C03625=1054.668,133.483,-83.506,171.485,33.116,156.194
C03626=1054.674,133.732,-83.526,171.487,33.118,156.195
C03627=1054.680,133.981,-83.548,171.489,33.121,156.195
C03628=1054.685,134.230,-83.568,171.490,33.123,156.195
C03629=1054.692,134.479,-83.589,171.492,33.125,156.196
C03630=1054.698,134.728,-83.610,171.494,33.128,156.196
C03631=1054.704,134.977,-83.632,171.496,33.130,156.197
C03632=1054.710,135.226,-83.652,171.498,33.132,156.197
C03633=1054.716,135.475,-83.673,171.499,33.135,156.197
C03634=1054.721,135.724,-83.694,171.501,33.137,156.198
C03635=1054.728,135.973,-83.715,171.503,33.139,156.198
C03636=1054.733,136.222,-83.735,171.505,33.142,156.199
C03637=1054.739,136.471,-83.757,171.507,33.145,156.199
C03638=1054.746,136.720,-83.778,171.508,33.146,156.199
C03639=1054.752,136.969,-83.799,171.510,33.149,156.200
C03640=1054.758,137.219,-83.820,171.512,33.152,156.200
C03641=1054.764,137.468,-83.840,171.514,33.154,156.201
C03642=1054.770,137.717,-83.862,171.516,33.156,156.201
C03643=1054.776,137.965,-83.883,171.518,33.159,156.201
C03644=1054.781,138.215,-83.904,171.519,33.161,156.202
C03645=1054.788,138.463,-83.925,171.521,33.163,156.202
C03646=1054.794,138.712,-83.946,171.523,33.166,156.203
C03647=1054.800,138.962,-83.967,171.525,33.168,156.203
C03648=1054.805,139.211,-83.989,171.527,33.170,156.203
C03649=1054.812,139.460,-84.010,171.528,33.173,156.204
C03650=1054.817,139.709,-84.030,171.530,33.175,156.204
C03651=1054.824,139.958,-84.052,171.532,33.178,156.205
C03652=1054.830,140.207,-84.073,171.534,33.180,156.205
C03653=1054.835,140.456,-84.094,171.536,33.183,156.205
C03654=1054.841,140.706,-84.116,171.538,33.185,156.206
C03655=1054.847,140.954,-84.137,171.539,33.188,156.206
C03656=1054.854,141.203,-84.158,171.541,33.190,156.207
C03657=1054.859,141.451,-84.179,171.543,33.192,156.207
C03658=1054.865,141.701,-84.200,171.545,33.195,156.207
C03659=1054.871,141.964,-84.223,171.547,33.197,156.208
C03660=1054.878,142.228,-84.246,171.549,33.200,156.208
C03661=1054.884,142.491,-84.268,171.551,33.203,156.209
C03662=1054.890,142.754,-84.291,171.553,33.205,156.209
C03663=1054.895,143.004,-84.312,171.554,33.208,156.210
C03664=1054.902,143.253,-84.333,171.556,33.210,156.210
C03665=1054.908,143.502,-84.355,171.558,33.212,156.210
C03666=1054.913,143.750,-84.376,171.560,33.215,156.211
C03667=1054.920,143.999,-84.397,171.562,33.217,156.211
C03668=1054.926,144.249,-84.419,171.564,33.220,156.212
C03669=1054.932,144.497,-84.440,171.566,33.222,156.212
C03670=1054.938,144.747,-84.461,171.567,33.224,156.212
C03671=1054.944,144.996,-84.483,171.569,33.227,156.213
C03672=1054.950,145.245,-84.504,171.571,33.229,156.213
C03673=1054.956,145.494,-84.526,171.573,33.231,156.214
C03674=1054.962,145.743,-84.547,171.575,33.234,156.214
C03675=1054.967,145.991,-84.568,171.577,33.237,156.214
C03676=1054.974,146.241,-84.590,171.579,33.239,156.215
C03677=1054.980,146.490,-84.612,171.580,33.241,156.215
C03678=1054.985,146.738,-84.633,171.582,33.244,156.216
C03679=1054.992,146.988,-84.655,171.584,33.246,156.216
C03680=1054.998,147.237,-84.676,171.586,33.249,156.217
C03681=1055.003,147.485,-84.698,171.588,33.251,156.217
C03682=1055.009,147.735,-84.719,171.590,33.253,156.217
C03683=1055.016,147.984,-84.741,171.592,33.256,156.218
C03684=1055.022,148.233,-84.762,171.593,33.258,156.218
C03685=1055.027,148.481,-84.784,171.595,33.261,156.219
C03686=1055.033,148.731,-84.805,171.597,33.263,156.219
C03687=1055.040,148.980,-84.827,171.599,33.266,156.219
C03688=1055.045,149.228,-84.848,171.601,33.268,156.220
C03689=1055.051,149.478,-84.870,171.603,33.271,156.220
C03690=1055.057,149.727,-84.892,171.605,33.273,156.221
C03691=1055.063,149.976,-84.914,171.607,33.276,156.221
C03692=1055.069,150.224,-84.936,171.608,33.278,156.221
C03693=1055.075,150.473,-84.957,171.610,33.280,156.222
C03694=1055.081,150.723,-84.979,171.612,33.283,156.222
C03695=1055.087,150.971,-85.000,171.614,33.285,156.223
C03696=1055.093,151.220,-85.022,171.616,33.288,156.223
C03697=1055.098,151.470,-85.044,171.618,33.291,156.224
C03698=1055.104,151.719,-85.066,171.620,33.292,156.224
C03699=1055.110,151.967,-85.088,171.622,33.295,156.224
C03700=1055.116,152.216,-85.109,171.624,33.298,156.225
C03701=1055.123,152.465,-85.131,171.625,33.300,156.225
C03702=1055.128,152.715,-85.153,171.627,33.303,156.226
C03703=1055.134,152.963,-85.175,171.629,33.305,156.226
C03704=1055.140,153.212,-85.197,171.632,33.308,156.227
C03705=1055.146,153.461,-85.219,171.634,33.310,156.227
C03706=1055.152,153.710,-85.240,171.636,33.312,156.227
C03707=1055.158,153.960,-85.262,171.638,33.315,156.228
C03708=1055.164,154.208,-85.284,171.640,33.317,156.228
C03709=1055.170,154.457,-85.306,171.642,33.320,156.229
C03710=1055.176,154.706,-85.328,171.644,33.323,156.229
C03711=1055.181,154.956,-85.350,171.645,33.324,156.229
C03712=1055.188,155.204,-85.372,171.647,33.327,156.230
C03713=1055.193,155.453,-85.394,171.649,33.330,156.230
C03714=1055.200,155.702,-85.415,171.651,33.332,156.231
C03715=1055.205,155.951,-85.438,171.653,33.335,156.231
C03716=1055.212,156.200,-85.460,171.655,33.337,156.232
C03717=1055.218,156.449,-85.481,171.657,33.340,156.232
C03718=1055.223,156.698,-85.504,171.659,33.342,156.233
C03719=1055.229,156.947,-85.526,171.661,33.345,156.233
C03720=1055.235,157.196,-85.549,171.663,33.348,156.233
C03721=1055.241,157.445,-85.570,171.665,33.350,156.234
C03722=1055.247,157.694,-85.592,171.667,33.352,156.234
C03723=1055.254,157.978,-85.617,171.669,33.355,156.235
C03724=1055.261,158.263,-85.642,171.671,33.358,156.235
C03725=1055.267,158.548,-85.668,171.673,33.361,156.236
C03726=1055.274,158.833,-85.693,171.675,33.364,156.236
C03727=1055.280,159.082,-85.715,171.677,33.366,156.237
C03728=1055.286,159.331,-85.738,171.679,33.369,156.237
C03729=1055.292,159.580,-85.760,171.681,33.371,156.237
C03730=1055.299,159.829,-85.782,171.683,33.374,156.238
C03731=1055.304,160.077,-85.804,171.685,33.376,156.238
C03732=1055.310,160.326,-85.826,171.687,33.379,156.239
C03733=1055.316,160.575,-85.849,171.689,33.381,156.239
C03734=1055.322,160.824,-85.870,171.691,33.383,156.240
C03735=1055.327,161.073,-85.893,171.693,33.387,156.240
C03736=1055.334,161.323,-85.915,171.695,33.389,156.241
C03737=1055.339,161.571,-85.938,171.697,33.392,156.241
C03738=1055.345,161.820,-85.961,171.699,33.394,156.241
C03739=1055.350,162.069,-85.983,171.701,33.397,156.242
C03740=1055.356,162.318,-86.005,171.703,33.399,156.242
C03741=1055.362,162.567,-86.028,171.705,33.402,156.243
C03742=1055.367,162.816,-86.050,171.706,33.404,156.243
C03743=1055.374,163.065,-86.073,171.708,33.407,156.244
C03744=1055.380,163.314,-86.096,171.710,33.410,156.244
C03745=1055.385,163.563,-86.118,171.712,33.413,156.245
C03746=1055.390,163.811,-86.140,171.714,33.415,156.245
C03747=1055.397,164.060,-86.163,171.716,33.418,156.245
C03748=1055.402,164.309,-86.185,171.718,33.420,156.246
C03749=1055.408,164.558,-86.208,171.720,33.423,156.246
C03750=1055.414,164.807,-86.231,171.723,33.425,156.247
C03751=1055.420,165.056,-86.253,171.725,33.428,156.247
C03752=1055.426,165.305,-86.275,171.727,33.431,156.248
C03753=1055.431,165.554,-86.298,171.729,33.433,156.248
C03754=1055.437,165.803,-86.321,171.731,33.436,156.249
C03755=1055.443,166.051,-86.343,171.733,33.439,156.249
C03756=1055.448,166.301,-86.366,171.735,33.441,156.250
C03757=1055.454,166.549,-86.389,171.737,33.444,156.250
C03758=1055.460,166.798,-86.411,171.739,33.446,156.250
C03759=1055.465,167.047,-86.434,171.741,33.449,156.251
C03760=1055.472,167.296,-86.457,171.743,33.452,156.251
C03761=1055.477,167.545,-86.479,171.745,33.454,156.252
C03762=1055.483,167.794,-86.502,171.747,33.457,156.252
C03763=1055.489,168.043,-86.525,171.749,33.459,156.253
C03764=1055.495,168.292,-86.547,171.751,33.462,156.253
C03765=1055.501,168.541,-86.570,171.753,33.465,156.254
C03766=1055.507,168.789,-86.593,171.755,33.468,156.254
C03767=1055.512,169.038,-86.616,171.757,33.470,156.255
C03768=1055.518,169.288,-86.638,171.759,33.473,156.255
C03769=1055.524,169.536,-86.661,171.761,33.475,156.255
C03770=1055.530,169.785,-86.684,171.763,33.478,156.256
C03771=1055.536,170.034,-86.707,171.765,33.480,156.256
C03772=1055.542,170.283,-86.729,171.767,33.483,156.257
C03773=1055.547,170.532,-86.752,171.769,33.485,156.257
C03774=1055.554,170.781,-86.775,171.771,33.488,156.258
C03775=1055.559,171.030,-86.798,171.773,33.491,156.258
C03776=1055.565,171.278,-86.821,171.775,33.494,156.259
C03777=1055.571,171.527,-86.844,171.777,33.496,156.259
C03778=1055.577,171.776,-86.867,171.779,33.499,156.260
C03779=1055.583,172.025,-86.889,171.781,33.501,156.260
C03780=1055.589,172.274,-86.912,171.783,33.504,156.260
C03781=1055.595,172.523,-86.935,171.785,33.506,156.261
C03782=1055.601,172.772,-86.958,171.788,33.509,156.261
C03783=1055.607,173.021,-86.981,171.790,33.511,156.262
C03784=1055.612,173.270,-87.004,171.792,33.514,156.262
C03785=1055.619,173.519,-87.026,171.794,33.517,156.263
C03786=1055.625,173.767,-87.049,171.796,33.520,156.263
C03787=1055.631,174.052,-87.076,171.798,33.522,156.264
C03788=1055.638,174.336,-87.102,171.801,33.525,156.264
C03789=1055.645,174.620,-87.128,171.803,33.529,156.265
C03790=1055.651,174.905,-87.155,171.805,33.531,156.265
C03791=1055.657,175.154,-87.178,171.808,33.534,156.266
C03792=1055.664,175.403,-87.200,171.810,33.537,156.266
C03793=1055.670,175.651,-87.224,171.812,33.539,156.267
C03794=1055.676,175.900,-87.247,171.814,33.542,156.267
C03795=1055.682,176.149,-87.270,171.816,33.545,156.267
C03796=1055.687,176.398,-87.293,171.818,33.547,156.268
C03797=1055.693,176.647,-87.316,171.820,33.550,156.268
C03798=1055.699,176.896,-87.339,171.822,33.552,156.269
C03799=1055.705,177.145,-87.363,171.824,33.555,156.269
C03800=1055.712,177.393,-87.385,171.826,33.558,156.270
C03801=1055.718,177.642,-87.408,171.828,33.560,156.270
C03802=1055.723,177.891,-87.431,171.830,33.563,156.271
C03803=1055.730,178.140,-87.455,171.832,33.565,156.271
C03804=1055.736,178.389,-87.478,171.834,33.568,156.272
C03805=1055.741,178.638,-87.501,171.837,33.571,156.272
C03806=1055.747,178.887,-87.524,171.839,33.573,156.272
C03807=1055.753,179.135,-87.548,171.841,33.576,156.273
C03808=1055.760,179.384,-87.570,171.844,33.579,156.273
C03809=1055.766,179.633,-87.593,171.846,33.581,156.274
C03810=1055.772,179.881,-87.617,171.848,33.584,156.274
C03811=1055.778,180.130,-87.640,171.850,33.586,156.275
C03812=1055.784,180.380,-87.663,171.852,33.589,156.275
C03813=1055.790,180.628,-87.687,171.854,33.592,156.276
C03814=1055.796,180.877,-87.710,171.856,33.594,156.276
C03815=1055.802,181.126,-87.733,171.859,33.597,156.277
C03816=1055.808,181.375,-87.757,171.861,33.600,156.277
C03817=1055.814,181.624,-87.780,171.863,33.602,156.278
C03818=1055.820,181.873,-87.803,171.865,33.605,156.278
C03819=1055.827,182.121,-87.826,171.867,33.607,156.278
C03820=1055.833,182.370,-87.849,171.869,33.610,156.279
C03821=1055.839,182.619,-87.873,171.871,33.613,156.279
C03822=1055.845,182.868,-87.896,171.873,33.615,156.280
C03823=1055.851,183.116,-87.920,171.876,33.618,156.280
C03824=1055.857,183.365,-87.943,171.878,33.621,156.281
C03825=1055.863,183.615,-87.966,171.880,33.623,156.281
C03826=1055.869,183.863,-87.989,171.882,33.626,156.282
C03827=1055.875,184.112,-88.012,171.884,33.628,156.282
C03828=1055.882,184.361,-88.036,171.886,33.631,156.283
C03829=1055.887,184.610,-88.059,171.888,33.634,156.283
C03830=1055.893,184.859,-88.084,171.892,33.637,156.284
C03831=1055.899,185.107,-88.107,171.894,33.640,156.284
C03832=1055.904,185.357,-88.131,171.896,33.642,156.285
C03833=1055.910,185.605,-88.155,171.898,33.645,156.285
C03834=1055.916,185.854,-88.179,171.900,33.648,156.286
C03835=1055.921,186.102,-88.202,171.902,33.651,156.286
C03836=1055.928,186.351,-88.226,171.904,33.654,156.287
C03837=1055.933,186.600,-88.250,171.906,33.656,156.287
C03838=1055.939,186.849,-88.273,171.909,33.659,156.288
C03839=1055.944,187.098,-88.298,171.911,33.662,156.288
C03840=1055.951,187.347,-88.322,171.913,33.664,156.288
C03841=1055.956,187.596,-88.345,171.915,33.668,156.289
C03842=1055.962,187.844,-88.369,171.917,33.670,156.289
C03843=1055.969,188.093,-88.393,171.919,33.673,156.290
C03844=1055.974,188.342,-88.416,171.921,33.676,156.290
C03845=1055.980,188.590,-88.440,171.923,33.679,156.291
C03846=1055.986,188.840,-88.465,171.926,33.682,156.291
C03847=1055.992,189.088,-88.488,171.928,33.685,156.292
C03848=1055.997,189.337,-88.513,171.931,33.687,156.292
C03849=1056.003,189.586,-88.536,171.933,33.690,156.293
C03850=1056.009,189.835,-88.560,171.935,33.693,156.294
C03851=1056.015,190.118,-88.588,171.938,33.696,156.294
C03852=1056.022,190.402,-88.615,171.940,33.699,156.295
C03853=1056.028,190.687,-88.642,171.943,33.702,156.295
C03854=1056.035,190.970,-88.670,171.945,33.705,156.296
C03855=1056.042,191.219,-88.694,171.947,33.709,156.296
C03856=1056.047,191.468,-88.718,171.950,33.711,156.297
C03857=1056.054,191.717,-88.742,171.952,33.714,156.297
C03858=1056.059,191.966,-88.765,171.954,33.717,156.298
C03859=1056.065,192.214,-88.789,171.956,33.720,156.298
C03860=1056.071,192.463,-88.813,171.958,33.722,156.299
C03861=1056.077,192.712,-88.837,171.960,33.726,156.299
C03862=1056.083,192.961,-88.861,171.963,33.728,156.300
C03863=1056.088,193.209,-88.886,171.965,33.731,156.300
C03864=1056.095,193.458,-88.909,171.967,33.734,156.301
C03865=1056.100,193.707,-88.934,171.970,33.737,156.301
C03866=1056.106,193.955,-88.958,171.972,33.739,156.302
C03867=1056.112,194.204,-88.982,171.975,33.742,156.302
C03868=1056.118,194.453,-89.006,171.977,33.745,156.303
C03869=1056.124,194.702,-89.030,171.979,33.748,156.303
C03870=1056.130,194.951,-89.055,171.981,33.751,156.304
C03871=1056.136,195.200,-89.079,171.984,33.753,156.304
C03872=1056.142,195.448,-89.103,171.986,33.757,156.305
C03873=1056.148,195.697,-89.127,171.988,33.759,156.305
C03874=1056.153,195.946,-89.151,171.990,33.762,156.306
C03875=1056.160,196.195,-89.175,171.992,33.765,156.306
C03876=1056.165,196.443,-89.200,171.995,33.768,156.307
C03877=1056.172,196.692,-89.224,171.997,33.771,156.307
C03878=1056.177,196.941,-89.248,171.999,33.774,156.308
C03879=1056.184,197.189,-89.273,172.001,33.777,156.308
C03880=1056.190,197.438,-89.297,172.005,33.779,156.309
C03881=1056.196,197.687,-89.321,172.007,33.782,156.309
C03882=1056.202,197.935,-89.345,172.009,33.785,156.310
C03883=1056.208,198.184,-89.369,172.011,33.788,156.310
C03884=1056.214,198.434,-89.394,172.014,33.791,156.311
C03885=1056.220,198.682,-89.419,172.016,33.794,156.311
C03886=1056.226,198.931,-89.443,172.018,33.796,156.312
C03887=1056.232,199.179,-89.467,172.020,33.799,156.312
C03888=1056.238,199.428,-89.491,172.023,33.802,156.313
C03889=1056.244,199.677,-89.515,172.025,33.805,156.313
C03890=1056.250,199.925,-89.540,172.027,33.808,156.314
C03891=1056.256,200.174,-89.565,172.030,33.811,156.314
C03892=1056.262,200.423,-89.589,172.032,33.813,156.315
C03893=1056.268,200.672,-89.613,172.034,33.816,156.316
C03894=1056.275,200.921,-89.638,172.037,33.819,156.316
C03895=1056.281,201.169,-89.662,172.040,33.822,156.317
C03896=1056.286,201.418,-89.687,172.042,33.825,156.317
C03897=1056.292,201.666,-89.712,172.044,33.828,156.318
C03898=1056.299,201.915,-89.736,172.047,33.831,156.318
C03899=1056.305,202.164,-89.760,172.049,33.834,156.319
C03900=1056.310,202.412,-89.785,172.051,33.836,156.319
C03901=1056.316,202.662,-89.810,172.053,33.840,156.320
C03902=1056.321,202.910,-89.834,172.056,33.843,156.320
C03903=1056.328,203.159,-89.859,172.058,33.845,156.321
C03904=1056.334,203.408,-89.883,172.060,33.848,156.321
C03905=1056.340,203.656,-89.908,172.063,33.852,156.322
C03906=1056.346,203.905,-89.933,172.065,33.855,156.322
C03907=1056.352,204.154,-89.958,172.067,33.857,156.323
C03908=1056.357,204.402,-89.983,172.070,33.860,156.323
C03909=1056.363,204.651,-90.008,172.073,33.863,156.324
C03910=1056.369,204.900,-90.032,172.075,33.866,156.325
C03911=1056.375,205.148,-90.058,172.077,33.870,156.325
C03912=1056.382,205.397,-90.082,172.080,33.872,156.326
C03913=1056.387,205.645,-90.107,172.082,33.875,156.326
C03914=1056.393,205.895,-90.131,172.084,33.878,156.327
C03915=1056.418,206.946,-90.237,172.283,33.968,156.339
C03916=1056.424,207.183,-90.261,172.285,33.972,156.340
C03917=1056.431,207.420,-90.286,172.287,33.975,156.341
C03918=1056.437,207.658,-90.310,172.288,33.979,156.342
C03919=1056.442,207.895,-90.336,172.291,33.983,156.342
C03920=1056.448,208.133,-90.360,172.293,33.986,156.343
C03921=1056.454,208.371,-90.384,172.295,33.990,156.344
C03922=1056.460,208.607,-90.409,172.296,33.993,156.344
C03923=1056.466,208.846,-90.434,172.298,33.997,156.345
C03924=1056.472,209.094,-90.460,172.300,34.001,156.346
C03925=1056.479,209.342,-90.485,172.302,34.005,156.347
C03926=1056.484,209.591,-90.512,172.304,34.009,156.347
C03927=1056.491,209.840,-90.537,172.306,34.013,156.348
C03928=1056.498,210.088,-90.564,172.308,34.017,156.349
C03929=1056.504,210.337,-90.589,172.310,34.020,156.349
C03930=1056.510,210.585,-90.616,172.312,34.024,156.350
C03931=1056.516,210.834,-90.641,172.314,34.028,156.351
C03932=1056.522,211.082,-90.667,172.315,34.032,156.352
C03933=1056.528,211.332,-90.693,172.317,34.035,156.352
C03934=1056.535,211.580,-90.719,172.320,34.040,156.353
C03935=1056.541,211.828,-90.745,172.322,34.043,156.354
C03936=1056.547,212.077,-90.771,172.324,34.047,156.355
C03937=1056.554,212.325,-90.798,172.326,34.051,156.355
C03938=1056.559,212.574,-90.824,172.327,34.055,156.356
C03939=1056.566,212.822,-90.850,172.329,34.058,156.357
C03940=1056.571,213.071,-90.876,172.332,34.062,156.358
C03941=1056.578,213.320,-90.902,172.334,34.066,156.358
C03942=1056.584,213.569,-90.929,172.336,34.070,156.359
C03943=1056.591,213.817,-90.954,172.338,34.074,156.360
C03944=1056.596,214.066,-90.981,172.339,34.078,156.361
C03945=1056.603,214.314,-91.007,172.341,34.081,156.361
C03946=1056.609,214.562,-91.033,172.343,34.085,156.362
C03947=1056.615,214.811,-91.059,172.346,34.089,156.363
C03948=1056.621,215.060,-91.086,172.348,34.093,156.363
C03949=1056.628,215.308,-91.112,172.350,34.097,156.364
C03950=1056.633,215.556,-91.138,172.352,34.100,156.365
C03951=1056.640,215.806,-91.164,172.354,34.104,156.366
C03952=1056.646,216.054,-91.191,172.355,34.108,156.366
C03953=1056.653,216.302,-91.217,172.357,34.112,156.367
C03954=1056.659,216.551,-91.244,172.360,34.115,156.368
C03955=1056.665,216.800,-91.269,172.362,34.119,156.368
C03956=1056.671,217.048,-91.296,172.364,34.123,156.369
C03957=1056.677,217.296,-91.322,172.366,34.127,156.370
C03958=1056.684,217.545,-91.349,172.368,34.130,156.371
C03959=1056.690,217.794,-91.376,172.370,34.134,156.371
C03960=1056.696,218.042,-91.402,172.373,34.138,156.372
C03961=1056.702,218.291,-91.428,172.374,34.142,156.373
C03962=1056.709,218.539,-91.454,172.376,34.146,156.374
C03963=1056.714,218.788,-91.481,172.378,34.149,156.374
C03964=1056.722,219.036,-91.507,172.380,34.153,156.375
C03965=1056.727,219.285,-91.534,172.382,34.156,156.376
C03966=1056.734,219.533,-91.560,172.384,34.161,156.377
C03967=1056.740,219.782,-91.587,172.387,34.164,156.377
C03968=1056.746,220.030,-91.613,172.389,34.168,156.378
C03969=1056.753,220.279,-91.640,172.391,34.172,156.379
C03970=1056.759,220.527,-91.666,172.393,34.175,156.379
C03971=1056.765,220.775,-91.692,172.395,34.179,156.380
C03972=1056.771,221.016,-91.718,172.397,34.183,156.381
C03973=1056.777,221.256,-91.744,172.399,34.186,156.382
C03974=1056.783,221.496,-91.769,172.401,34.190,156.382
C03975=1056.789,221.736,-91.795,172.403,34.194,156.383
C03976=1056.795,221.976,-91.822,172.405,34.198,156.384
C03977=1056.801,222.217,-91.847,172.407,34.201,156.384
C03978=1056.808,222.457,-91.873,172.409,34.205,156.385
C03979=1056.813,222.697,-91.899,172.412,34.209,156.386
C03980=1056.819,222.945,-91.926,172.413,34.212,156.387
C03981=1056.825,223.193,-91.952,172.415,34.216,156.387
C03982=1056.831,223.442,-91.979,172.417,34.219,156.388
C03983=1056.837,223.691,-92.006,172.419,34.223,156.389
C03984=1056.844,223.940,-92.032,172.421,34.227,156.389
C03985=1056.850,224.188,-92.059,172.424,34.231,156.390
C03986=1056.857,224.436,-92.087,172.426,34.235,156.391
C03987=1056.863,224.685,-92.113,172.428,34.238,156.392
C03988=1056.868,224.933,-92.140,172.430,34.242,156.392
C03989=1056.875,225.182,-92.167,172.432,34.246,156.393
C03990=1056.881,225.430,-92.193,172.434,34.250,156.394
C03991=1056.888,225.679,-92.221,172.437,34.253,156.395
C03992=1056.894,225.927,-92.248,172.439,34.257,156.395
C03993=1056.900,226.176,-92.275,172.441,34.261,156.396
C03994=1056.906,226.424,-92.301,172.443,34.264,156.397
C03995=1056.912,226.673,-92.329,172.445,34.268,156.397
C03996=1056.919,226.921,-92.355,172.447,34.272,156.398
C03997=1056.925,227.170,-92.382,172.450,34.276,156.399
C03998=1056.931,227.418,-92.409,172.452,34.279,156.400
C03999=1056.938,227.667,-92.436,172.454,34.283,156.400
C04000=1056.944,227.915,-92.463,172.456,34.287,156.401
C04001=1056.950,228.164,-92.491,172.458,34.290,156.402
C04002=1056.956,228.412,-92.517,172.460,34.294,156.402
C04003=1056.963,228.661,-92.544,172.463,34.298,156.403
C04004=1056.969,228.908,-92.571,172.465,34.302,156.404
C04005=1056.976,229.157,-92.598,172.467,34.305,156.405
C04006=1056.981,229.406,-92.625,172.469,34.309,156.405
C04007=1056.988,229.654,-92.653,172.471,34.313,156.406
C04008=1056.994,229.903,-92.679,172.473,34.316,156.407
C04009=1057.001,230.151,-92.707,172.476,34.320,156.407
C04010=1057.006,230.399,-92.734,172.478,34.324,156.408
C04011=1057.013,230.648,-92.761,172.480,34.328,156.409
C04012=1057.019,230.897,-92.789,172.482,34.331,156.410
C04013=1057.025,231.145,-92.816,172.484,34.335,156.410
C04014=1057.031,231.394,-92.843,172.487,34.339,156.411
C04015=1057.037,231.642,-92.871,172.489,34.342,156.412
C04016=1057.044,231.891,-92.898,172.491,34.346,156.413
C04017=1057.050,232.139,-92.925,172.493,34.350,156.413
C04018=1057.056,232.388,-92.952,172.495,34.354,156.414
C04019=1057.062,232.635,-92.979,172.497,34.357,156.415
C04020=1057.068,232.884,-93.006,172.500,34.361,156.416
C04021=1057.075,233.133,-93.034,172.502,34.364,156.416
C04022=1057.080,233.381,-93.062,172.504,34.368,156.417
C04023=1057.087,233.630,-93.089,172.506,34.372,156.418
C04024=1057.093,233.878,-93.117,172.508,34.376,156.418
C04025=1057.100,234.126,-93.144,172.512,34.380,156.419
C04026=1057.105,234.375,-93.172,172.514,34.383,156.420
C04027=1057.111,234.623,-93.199,172.516,34.387,156.421
C04028=1057.117,234.860,-93.225,172.518,34.390,156.421
C04029=1057.124,235.096,-93.252,172.520,34.394,156.422
C04030=1057.129,235.332,-93.278,172.522,34.398,156.423
C04031=1057.135,235.568,-93.304,172.524,34.401,156.423
C04032=1057.141,235.804,-93.330,172.526,34.405,156.424
C04033=1057.147,236.041,-93.357,172.528,34.408,156.425
C04034=1057.153,236.277,-93.382,172.530,34.412,156.425
C04035=1057.159,236.513,-93.409,172.532,34.415,156.426
C04036=1057.165,236.762,-93.436,172.535,34.419,156.427
C04037=1057.171,237.010,-93.464,172.538,34.422,156.428
C04038=1057.177,237.258,-93.491,172.540,34.426,156.428
C04039=1057.184,237.507,-93.519,172.542,34.430,156.429
C04040=1057.190,237.754,-93.547,172.544,34.434,156.430
C04041=1057.196,238.003,-93.575,172.546,34.437,156.430
C04042=1057.202,238.252,-93.602,172.549,34.441,156.431
C04043=1057.208,238.500,-93.629,172.551,34.445,156.432
C04044=1057.215,238.748,-93.657,172.553,34.448,156.433
C04045=1057.221,238.997,-93.685,172.555,34.452,156.433
C04046=1057.228,239.245,-93.713,172.557,34.456,156.434
C04047=1057.234,239.493,-93.740,172.561,34.459,156.435
C04048=1057.240,239.742,-93.769,172.563,34.463,156.435
C04049=1057.246,239.990,-93.796,172.565,34.466,156.436
C04050=1057.253,240.239,-93.824,172.567,34.471,156.437
C04051=1057.258,240.487,-93.852,172.569,34.474,156.438
C04052=1057.265,240.735,-93.880,172.572,34.478,156.438
C04053=1057.272,240.984,-93.908,172.574,34.481,156.439
C04054=1057.278,241.233,-93.936,172.576,34.485,156.440
C04055=1057.284,241.480,-93.963,172.579,34.489,156.441
C04056=1057.290,241.729,-93.991,172.581,34.492,156.441
C04057=1057.296,241.977,-94.019,172.584,34.496,156.442
C04058=1057.303,242.226,-94.047,172.586,34.500,156.443
C04059=1057.308,242.474,-94.075,172.588,34.503,156.443
C04060=1057.315,242.722,-94.103,172.590,34.507,156.444
C04061=1057.321,242.971,-94.131,172.592,34.511,156.445
C04062=1057.327,243.220,-94.159,172.596,34.515,156.446
C04063=1057.333,243.468,-94.187,172.598,34.518,156.446
C04064=1057.339,243.716,-94.215,172.600,34.522,156.447
C04065=1057.346,243.964,-94.244,172.602,34.525,156.448
C04066=1057.352,244.213,-94.272,172.604,34.529,156.448
C04067=1057.358,244.461,-94.299,172.607,34.533,156.449
C04068=1057.364,244.709,-94.328,172.609,34.537,156.450
C04069=1057.370,244.958,-94.356,172.612,34.540,156.451
C04070=1057.377,245.206,-94.384,172.614,34.544,156.451
C04071=1057.383,245.455,-94.413,172.616,34.548,156.452
C04072=1057.390,245.703,-94.440,172.619,34.551,156.453
C04073=1057.395,245.951,-94.468,172.621,34.555,156.454
C04074=1057.401,246.200,-94.497,172.623,34.558,156.454
C04075=1057.408,246.448,-94.525,172.626,34.563,156.455
C04076=1057.414,246.697,-94.553,172.628,34.566,156.456
C04077=1057.420,246.945,-94.582,172.631,34.570,156.457
C04078=1057.425,247.193,-94.610,172.633,34.574,156.457
C04079=1057.432,247.441,-94.638,172.635,34.577,156.458
C04080=1057.438,247.689,-94.667,172.637,34.581,156.459
C04081=1057.444,247.938,-94.696,172.641,34.585,156.460
C04082=1057.450,248.187,-94.724,172.643,34.589,156.460
C04083=1057.456,248.434,-94.753,172.645,34.592,156.461
C04084=1057.462,248.668,-94.779,172.647,34.596,156.462
C04085=1057.468,248.901,-94.806,172.649,34.599,156.462
C04086=1057.473,249.134,-94.833,172.652,34.603,156.463
C04087=1057.479,249.367,-94.859,172.654,34.607,156.464
C04088=1057.485,249.600,-94.886,172.656,34.610,156.464
C04089=1057.491,249.834,-94.912,172.658,34.613,156.465
C04090=1057.496,250.067,-94.940,172.660,34.617,156.466
C04091=1057.502,250.300,-94.967,172.664,34.620,156.467
C04092=1057.508,250.548,-94.995,172.666,34.624,156.467
C04093=1057.514,250.797,-95.024,172.668,34.628,156.468
C04094=1057.520,251.045,-95.052,172.670,34.631,156.469
C04095=1057.527,251.293,-95.081,172.672,34.635,156.469
C04096=1057.533,251.542,-95.109,172.676,34.639,156.470
C04097=1057.539,251.789,-95.138,172.678,34.643,156.471
C04098=1057.545,252.037,-95.167,172.680,34.646,156.472
C04099=1057.551,252.286,-95.195,172.682,34.650,156.472
C04100=1057.557,252.534,-95.224,172.686,34.653,156.473
C04101=1057.563,252.783,-95.253,172.688,34.657,156.474
C04102=1057.570,253.031,-95.281,172.690,34.661,156.475
C04103=1057.577,253.279,-95.310,172.692,34.665,156.475
C04104=1057.583,253.528,-95.338,172.695,34.668,156.476
C04105=1057.589,253.776,-95.367,172.698,34.672,156.477
C04106=1057.595,254.024,-95.396,172.700,34.676,156.478
C04107=1057.601,254.273,-95.425,172.702,34.679,156.478
C04108=1057.607,254.521,-95.454,172.705,34.683,156.479
C04109=1057.613,254.769,-95.483,172.708,34.686,156.480
C04110=1057.620,255.017,-95.512,172.710,34.690,156.480
C04111=1057.626,255.266,-95.540,172.712,34.694,156.481
C04112=1057.633,255.514,-95.569,172.715,34.698,156.482
C04113=1057.639,255.762,-95.598,172.717,34.701,156.483
C04114=1057.645,256.010,-95.627,172.720,34.705,156.483
C04115=1057.651,256.258,-95.656,172.723,34.709,156.484
C04116=1057.657,256.507,-95.684,172.725,34.712,156.485
C04117=1057.664,256.755,-95.713,172.727,34.716,156.486
C04118=1057.670,257.003,-95.742,172.730,34.719,156.486
C04119=1057.676,257.251,-95.771,172.733,34.723,156.487
C04120=1057.683,257.500,-95.801,172.735,34.727,156.488
C04121=1057.689,257.748,-95.830,172.737,34.730,156.488
C04122=1057.696,257.997,-95.857,172.740,34.734,156.489
C04123=1057.702,258.245,-95.886,172.743,34.738,156.490
C04124=1057.708,258.493,-95.915,172.745,34.741,156.491
C04125=1057.715,258.741,-95.944,172.748,34.745,156.491
C04126=1057.721,258.989,-95.974,172.750,34.749,156.492
C04127=1057.727,259.237,-96.003,172.753,34.752,156.493
C04128=1057.733,259.485,-96.032,172.756,34.756,156.494
C04129=1057.740,259.734,-96.061,172.758,34.759,156.494
C04130=1057.746,259.982,-96.090,172.760,34.763,156.495
C04131=1057.753,260.231,-96.119,172.764,34.767,156.496
C04132=1057.759,260.479,-96.148,172.766,34.770,156.496
C04133=1057.765,260.727,-96.177,172.768,34.774,156.497
C04134=1057.771,260.975,-96.206,172.771,34.777,156.498
C04135=1057.778,261.224,-96.236,172.773,34.781,156.499
C04136=1057.785,261.472,-96.265,172.776,34.785,156.499
C04137=1057.791,261.720,-96.294,172.779,34.788,156.500
C04138=1057.797,261.968,-96.323,172.781,34.792,156.501
C04139=1057.803,262.216,-96.352,172.784,34.795,156.501
C04140=1057.810,262.448,-96.379,172.787,34.799,156.502
C04141=1057.816,262.680,-96.407,172.789,34.803,156.503
C04142=1057.822,262.912,-96.434,172.791,34.806,156.503
C04143=1057.828,263.145,-96.461,172.793,34.809,156.504
C04144=1057.834,263.378,-96.489,172.797,34.813,156.505
C04145=1057.840,263.610,-96.517,172.799,34.816,156.506
C04146=1057.846,263.841,-96.544,172.801,34.819,156.506
C04147=1057.851,264.073,-96.572,172.803,34.823,156.507
C04148=1057.857,264.321,-96.601,172.806,34.827,156.508
C04149=1057.864,264.570,-96.630,172.809,34.831,156.509
C04150=1057.870,264.819,-96.660,172.811,34.834,156.509
C04151=1057.876,265.066,-96.690,172.814,34.838,156.510
C04152=1057.882,265.314,-96.719,172.816,34.841,156.511
C04153=1057.888,265.563,-96.748,172.820,34.845,156.511
C04154=1057.895,265.811,-96.779,172.822,34.849,156.512
C04155=1057.901,266.059,-96.808,172.824,34.853,156.513
C04156=1057.907,266.308,-96.837,172.827,34.856,156.514
C04157=1057.913,266.555,-96.867,172.830,34.860,156.514
C04158=1057.920,266.804,-96.896,172.833,34.864,156.515
C04159=1057.926,267.052,-96.927,172.835,34.867,156.516
C04160=1057.932,267.300,-96.956,172.837,34.871,156.517
C04161=1057.939,267.548,-96.985,172.841,34.875,156.517
C04162=1057.945,267.797,-97.016,172.843,34.878,156.518
C04163=1057.951,268.045,-97.045,172.846,34.882,156.519
C04164=1057.958,268.292,-97.074,172.848,34.886,156.520
C04165=1057.963,268.541,-97.104,172.851,34.890,156.520
C04166=1057.971,268.789,-97.134,172.854,34.893,156.521
C04167=1057.976,269.037,-97.164,172.856,34.897,156.522
C04168=1057.983,269.285,-97.194,172.859,34.900,156.523
C04169=1057.989,269.534,-97.223,172.862,34.904,156.523
C04170=1057.995,269.781,-97.253,172.865,34.908,156.524
C04171=1058.002,270.029,-97.283,172.867,34.912,156.525
C04172=1058.008,270.278,-97.313,172.869,34.915,156.526
C04173=1058.014,270.526,-97.343,172.873,34.919,156.526
C04174=1058.020,270.774,-97.372,172.875,34.923,156.527
C04175=1058.027,271.022,-97.403,172.878,34.927,156.528
C04176=1058.033,271.270,-97.433,172.881,34.930,156.529
C04177=1058.039,271.518,-97.462,172.884,34.934,156.529
C04178=1058.046,271.767,-97.493,172.886,34.937,156.530
C04179=1058.052,272.014,-97.522,172.889,34.942,156.531
C04180=1058.058,272.262,-97.553,172.892,34.945,156.532
C04181=1058.065,272.511,-97.582,172.895,34.949,156.532
C04182=1058.071,272.759,-97.613,172.897,34.952,156.533
C04183=1058.076,273.007,-97.643,172.899,34.956,156.534
C04184=1058.084,273.255,-97.673,172.903,34.960,156.535
C04185=1058.089,273.503,-97.703,172.905,34.964,156.535
C04186=1058.095,273.751,-97.733,172.908,34.967,156.536
C04187=1058.102,273.999,-97.763,172.910,34.971,156.537
C04188=1058.108,274.247,-97.793,172.914,34.975,156.538
C04189=1058.115,274.495,-97.824,172.916,34.978,156.538
C04190=1058.121,274.743,-97.854,172.919,34.983,156.539
C04191=1058.126,274.991,-97.884,172.922,34.986,156.540
C04192=1058.134,275.240,-97.914,172.925,34.990,156.541
C04193=1058.139,275.488,-97.944,172.927,34.993,156.541
C04194=1058.146,275.736,-97.975,172.930,34.997,156.542
C04195=1058.152,275.984,-98.005,172.933,35.001,156.543
C04196=1058.158,276.218,-98.033,172.936,35.005,156.544
C04197=1058.163,276.452,-98.062,172.938,35.008,156.544
C04198=1058.170,276.686,-98.090,172.940,35.012,156.545
C04199=1058.176,276.920,-98.120,172.944,35.015,156.546
C04200=1058.182,277.155,-98.148,172.946,35.019,156.547
C04201=1058.188,277.388,-98.177,172.949,35.022,156.547
C04202=1058.193,277.623,-98.206,172.951,35.026,156.548
C04203=1058.200,277.857,-98.234,172.954,35.030,156.549
C04204=1058.206,278.105,-98.264,172.957,35.033,156.550
C04205=1058.212,278.353,-98.296,172.959,35.037,156.550
C04206=1058.218,278.601,-98.326,172.962,35.040,156.551
C04207=1058.225,278.849,-98.356,172.965,35.044,156.552
C04208=1058.231,279.097,-98.386,172.968,35.048,156.553
C04209=1058.237,279.345,-98.417,172.970,35.052,156.553
C04210=1058.243,279.593,-98.448,172.974,35.056,156.554
C04211=1058.250,279.841,-98.478,172.977,35.059,156.555
C04212=1058.256,280.089,-98.508,172.979,35.063,156.556
C04213=1058.263,280.337,-98.539,172.982,35.067,156.556
C04214=1058.269,280.585,-98.570,172.985,35.070,156.557
C04215=1058.275,280.833,-98.601,172.988,35.074,156.558
C04216=1058.281,281.081,-98.631,172.990,35.078,156.559
C04217=1058.288,281.329,-98.662,172.994,35.082,156.559
C04218=1058.294,281.577,-98.693,172.996,35.086,156.560
C04219=1058.300,281.825,-98.723,172.999,35.089,156.561
C04220=1058.306,282.073,-98.754,173.003,35.094,156.562
C04221=1058.313,282.321,-98.785,173.005,35.097,156.563
C04222=1058.318,282.569,-98.815,173.008,35.101,156.563
C04223=1058.325,282.817,-98.847,173.010,35.105,156.564
C04224=1058.332,283.065,-98.878,173.014,35.108,156.565
C04225=1058.337,283.313,-98.908,173.016,35.113,156.566
C04226=1058.344,283.561,-98.939,173.019,35.116,156.567
C04227=1058.350,283.809,-98.970,173.023,35.120,156.567
C04228=1058.357,284.057,-99.001,173.025,35.124,156.568
C04229=1058.363,284.305,-99.032,173.028,35.127,156.569
C04230=1058.369,284.553,-99.062,173.030,35.131,156.570
C04231=1058.376,284.801,-99.094,173.034,35.135,156.570
C04232=1058.381,285.049,-99.124,173.037,35.139,156.571
C04233=1058.388,285.297,-99.155,173.039,35.143,156.572
C04234=1058.395,285.545,-99.186,173.043,35.146,156.573
C04235=1058.401,285.793,-99.217,173.046,35.150,156.574
C04236=1058.407,286.041,-99.248,173.048,35.154,156.574
C04237=1058.414,286.289,-99.279,173.052,35.158,156.575
C04238=1058.420,286.536,-99.310,173.054,35.162,156.576
C04239=1058.426,286.785,-99.341,173.057,35.165,156.577
C04240=1058.433,287.033,-99.373,173.060,35.169,156.577
C04241=1058.438,287.281,-99.404,173.063,35.173,156.578
C04242=1058.445,287.529,-99.435,173.066,35.177,156.579
C04243=1058.452,287.777,-99.466,173.069,35.181,156.580
C04244=1058.458,288.025,-99.497,173.072,35.184,156.581
C04245=1058.464,288.272,-99.528,173.075,35.188,156.581
C04246=1058.471,288.520,-99.560,173.078,35.192,156.582
C04247=1058.477,288.769,-99.590,173.081,35.196,156.583
C04248=1058.483,289.016,-99.621,173.084,35.199,156.584
C04249=1058.489,289.264,-99.653,173.087,35.204,156.585
C04250=1058.496,289.512,-99.685,173.090,35.207,156.585
C04251=1058.503,289.761,-99.716,173.093,35.211,156.586
C04252=1058.509,289.999,-99.746,173.095,35.215,156.587
C04253=1058.515,290.239,-99.776,173.098,35.218,156.588
C04254=1058.520,290.479,-99.807,173.102,35.222,156.588
C04255=1058.527,290.719,-99.837,173.104,35.226,156.589
C04256=1058.533,290.958,-99.868,173.107,35.230,156.590
C04257=1058.539,291.197,-99.898,173.110,35.234,156.591
C04258=1058.545,291.437,-99.928,173.113,35.237,156.592
C04259=1058.551,291.676,-99.959,173.116,35.241,156.592
C04260=1058.558,291.924,-99.991,173.119,35.245,156.593
C04261=1058.564,292.172,-100.021,173.122,35.249,156.594
C04262=1058.570,292.420,-100.052,173.125,35.252,156.595
C04263=1058.576,292.668,-100.084,173.128,35.257,156.596
C04264=1058.583,292.916,-100.116,173.131,35.260,156.596
C04265=1058.589,293.164,-100.148,173.134,35.264,156.597
C04266=1058.596,293.412,-100.179,173.137,35.268,156.598
C04267=1058.602,293.659,-100.210,173.140,35.272,156.599
C04268=1058.608,293.908,-100.242,173.143,35.276,156.600
C04269=1058.615,294.156,-100.274,173.147,35.280,156.600
C04270=1058.622,294.403,-100.306,173.149,35.284,156.601
C04271=1058.628,294.651,-100.338,173.152,35.287,156.602
C04272=1058.634,294.899,-100.370,173.156,35.291,156.603
C04273=1058.640,295.146,-100.401,173.159,35.295,156.604
C04274=1058.646,295.394,-100.433,173.161,35.299,156.604
C04275=1058.653,295.642,-100.464,173.165,35.303,156.605
C04276=1058.659,295.891,-100.496,173.168,35.307,156.606
C04277=1058.666,296.138,-100.527,173.170,35.311,156.607
C04278=1058.672,296.386,-100.560,173.174,35.315,156.608
C04279=1058.679,296.634,-100.592,173.177,35.318,156.608
C04280=1058.685,296.882,-100.624,173.180,35.322,156.609
C04281=1058.690,297.130,-100.655,173.183,35.327,156.610
C04282=1058.697,297.377,-100.687,173.186,35.331,156.611
C04283=1058.703,297.625,-100.720,173.189,35.335,156.612
C04284=1058.709,297.873,-100.752,173.193,35.338,156.613
C04285=1058.716,298.121,-100.784,173.195,35.342,156.614
C04286=1058.722,298.369,-100.816,173.198,35.347,156.614
C04287=1058.728,298.617,-100.848,173.202,35.351,156.615
C04288=1058.734,298.864,-100.880,173.205,35.355,156.616
C04289=1058.740,299.112,-100.912,173.207,35.359,156.617
C04290=1058.747,299.359,-100.944,173.211,35.362,156.618
C04291=1058.753,299.608,-100.976,173.214,35.366,156.619
C04292=1058.759,299.855,-101.009,173.217,35.371,156.619
C04293=1058.765,300.103,-101.041,173.221,35.375,156.620
C04294=1058.771,300.351,-101.074,173.223,35.379,156.621
C04295=1058.778,300.599,-101.105,173.227,35.383,156.622
C04296=1058.785,300.847,-101.138,173.230,35.386,156.623
C04297=1058.790,301.095,-101.170,173.233,35.390,156.624
C04298=1058.797,301.342,-101.203,173.237,35.395,156.624
C04299=1058.803,301.591,-101.235,173.239,35.399,156.625
C04300=1058.810,301.838,-101.267,173.242,35.403,156.626
C04301=1058.816,302.086,-101.299,173.246,35.407,156.627
C04302=1058.822,302.334,-101.332,173.249,35.410,156.628
C04303=1058.828,302.581,-101.364,173.252,35.414,156.629
C04304=1058.834,302.829,-101.397,173.255,35.419,156.630
C04305=1058.841,303.077,-101.429,173.258,35.423,156.630
C04306=1058.848,303.324,-101.461,173.261,35.427,156.631
C04307=1058.854,303.573,-101.493,173.265,35.431,156.632
C04308=1058.864,303.971,-101.546,173.269,35.437,156.633
C04309=1058.873,304.369,-101.598,173.275,35.444,156.635
C04310=1058.882,304.664,-101.636,173.278,35.448,156.636
C04311=1058.889,304.959,-101.676,173.283,35.453,156.637
C04312=1058.897,305.255,-101.715,173.286,35.458,156.638
C04313=1058.904,305.550,-101.752,173.291,35.463,156.639
C04314=1058.911,305.798,-101.785,173.294,35.467,156.640
C04315=1058.918,306.046,-101.818,173.297,35.471,156.641
C04316=1058.924,306.294,-101.851,173.300,35.475,156.642
C04317=1058.930,306.541,-101.884,173.303,35.479,156.642
C04318=1058.937,306.789,-101.917,173.307,35.483,156.643
C04319=1058.944,307.036,-101.949,173.310,35.487,156.644
C04320=1058.950,307.284,-101.981,173.313,35.491,156.645
C04321=1058.956,307.533,-102.014,173.317,35.495,156.646
C04322=1058.963,307.780,-102.047,173.320,35.499,156.647
C04323=1058.969,308.028,-102.079,173.324,35.503,156.647
C04324=1058.975,308.275,-102.112,173.327,35.507,156.648
C04325=1058.982,308.523,-102.145,173.329,35.511,156.649
C04326=1058.988,308.771,-102.178,173.333,35.515,156.650
C04327=1058.995,309.019,-102.211,173.336,35.520,156.651
C04328=1059.002,309.266,-102.243,173.339,35.524,156.652
C04329=1059.008,309.514,-102.276,173.343,35.528,156.653
C04330=1059.015,309.761,-102.309,173.346,35.532,156.654
C04331=1059.022,310.009,-102.342,173.350,35.536,156.654
C04332=1059.028,310.257,-102.375,173.353,35.540,156.655
C04333=1059.034,310.504,-102.408,173.356,35.544,156.656
C04334=1059.041,310.753,-102.441,173.360,35.548,156.657
C04335=1059.047,311.000,-102.473,173.363,35.552,156.658
C04336=1059.054,311.248,-102.506,173.367,35.556,156.659
C04337=1059.061,311.496,-102.539,173.370,35.560,156.660
C04338=1059.067,311.743,-102.573,173.373,35.564,156.661
C04339=1059.073,311.991,-102.606,173.377,35.568,156.661
C04340=1059.080,312.239,-102.639,173.380,35.573,156.662
C04341=1059.087,312.486,-102.671,173.384,35.577,156.663
C04342=1059.094,312.734,-102.704,173.387,35.581,156.664
C04343=1059.101,312.981,-102.737,173.390,35.585,156.665
C04344=1059.107,313.229,-102.770,173.394,35.589,156.666
C04345=1059.114,313.477,-102.803,173.397,35.593,156.667
C04346=1059.121,313.724,-102.837,173.401,35.597,156.667
C04347=1059.126,313.972,-102.870,173.403,35.601,156.668
C04348=1059.133,314.220,-102.903,173.406,35.606,156.669
C04349=1059.139,314.468,-102.937,173.410,35.610,156.670
C04350=1059.145,314.715,-102.970,173.413,35.614,156.671
C04351=1059.152,314.963,-103.004,173.417,35.618,156.672
C04352=1059.158,315.211,-103.037,173.420,35.622,156.673
C04353=1059.164,315.458,-103.071,173.423,35.627,156.674
C04354=1059.171,315.707,-103.104,173.427,35.631,156.675
C04355=1059.177,315.954,-103.138,173.430,35.635,156.676
C04356=1059.183,316.201,-103.171,173.434,35.639,156.677
C04357=1059.189,316.449,-103.205,173.437,35.644,156.678
C04358=1059.196,316.696,-103.239,173.441,35.648,156.678
C04359=1059.202,316.944,-103.272,173.444,35.653,156.679
C04360=1059.209,317.192,-103.306,173.447,35.657,156.680
C04361=1059.215,317.439,-103.340,173.451,35.661,156.681
C04362=1059.222,317.690,-103.374,173.454,35.665,156.682
C04363=1059.228,317.941,-103.408,173.458,35.669,156.683
C04364=1059.234,318.192,-103.442,173.461,35.674,156.684
C04365=1059.241,318.443,-103.476,173.465,35.678,156.685
C04366=1059.247,318.690,-103.510,173.468,35.683,156.686
C04367=1059.254,318.938,-103.543,173.472,35.687,156.687
C04368=1059.260,319.185,-103.577,173.475,35.691,156.688
C04369=1059.267,319.433,-103.611,173.478,35.695,156.689
C04370=1059.273,319.681,-103.645,173.483,35.700,156.690
C04371=1059.280,319.929,-103.678,173.486,35.704,156.691
C04372=1059.286,320.176,-103.712,173.490,35.709,156.692
C04373=1059.292,320.424,-103.747,173.493,35.713,156.692
C04374=1059.299,320.671,-103.780,173.497,35.717,156.693
C04375=1059.305,320.919,-103.814,173.500,35.721,156.694
C04376=1059.312,321.166,-103.847,173.503,35.725,156.695
C04377=1059.318,321.414,-103.882,173.507,35.730,156.696
C04378=1059.325,321.662,-103.916,173.510,35.734,156.697
C04379=1059.331,321.909,-103.950,173.514,35.739,156.698
C04380=1059.338,322.157,-103.984,173.517,35.743,156.699
C04381=1059.344,322.404,-104.018,173.521,35.747,156.700
C04382=1059.351,322.652,-104.052,173.524,35.752,156.701
C04383=1059.358,322.900,-104.086,173.528,35.756,156.702
C04384=1059.364,323.147,-104.120,173.532,35.761,156.703
C04385=1059.371,323.395,-104.154,173.536,35.765,156.704
C04386=1059.377,323.642,-104.188,173.539,35.769,156.705
C04387=1059.384,323.890,-104.222,173.543,35.773,156.706
C04388=1059.390,324.138,-104.256,173.546,35.778,156.707
C04389=1059.396,324.385,-104.290,173.549,35.782,156.708
C04390=1059.403,324.633,-104.324,173.553,35.787,156.709
C04391=1059.410,324.881,-104.358,173.556,35.791,156.710
C04392=1059.417,325.128,-104.393,173.560,35.795,156.710
C04393=1059.423,325.375,-104.427,173.564,35.800,156.711
C04394=1059.430,325.623,-104.461,173.568,35.804,156.712
C04395=1059.437,325.871,-104.495,173.571,35.809,156.713
C04396=1059.443,326.119,-104.530,173.575,35.813,156.714
C04397=1059.450,326.366,-104.564,173.578,35.817,156.715
C04398=1059.457,326.613,-104.598,173.582,35.822,156.716
C04399=1059.463,326.861,-104.633,173.586,35.826,156.717
C04400=1059.470,327.109,-104.666,173.590,35.830,156.718
C04401=1059.477,327.355,-104.701,173.593,35.835,156.719
C04402=1059.483,327.603,-104.736,173.597,35.840,156.720
C04403=1059.490,327.851,-104.769,173.600,35.844,156.721
C04404=1059.497,328.099,-104.805,173.604,35.848,156.722
C04405=1059.503,328.347,-104.839,173.608,35.853,156.723
C04406=1059.511,328.594,-104.873,173.611,35.857,156.724
C04407=1059.517,328.841,-104.908,173.615,35.861,156.725
C04408=1059.523,329.089,-104.942,173.619,35.866,156.726
C04409=1059.531,329.336,-104.977,173.622,35.871,156.727
C04410=1059.537,329.584,-105.011,173.626,35.875,156.728
C04411=1059.544,329.832,-105.045,173.630,35.879,156.729
C04412=1059.551,330.079,-105.080,173.633,35.884,156.730
C04413=1059.558,330.327,-105.114,173.637,35.888,156.731
C04414=1059.564,330.574,-105.150,173.641,35.892,156.732
C04415=1059.571,330.822,-105.185,173.645,35.897,156.733
C04416=1059.577,331.069,-105.219,173.648,35.902,156.734
C04417=1059.584,331.316,-105.254,173.652,35.906,156.735
C04418=1059.590,331.563,-105.289,173.655,35.911,156.736
C04419=1059.597,331.809,-105.323,173.660,35.915,156.737
C04420=1059.603,332.056,-105.358,173.663,35.920,156.738
C04421=1059.610,332.302,-105.392,173.667,35.924,156.739
C04422=1059.616,332.548,-105.427,173.671,35.929,156.740
C04423=1059.623,332.795,-105.462,173.674,35.934,156.741
C04424=1059.630,333.041,-105.497,173.679,35.938,156.742
C04425=1059.637,333.288,-105.532,173.682,35.943,156.743
C04426=1059.643,333.535,-105.567,173.686,35.947,156.744
C04427=1059.650,333.782,-105.602,173.689,35.952,156.745
C04428=1059.656,334.030,-105.636,173.694,35.957,156.746
C04429=1059.663,334.277,-105.671,173.697,35.962,156.747
C04430=1059.670,334.525,-105.707,173.701,35.966,156.748
C04431=1059.676,334.772,-105.742,173.705,35.971,156.749
C04432=1059.682,335.020,-105.777,173.709,35.975,156.750
C04433=1059.689,335.267,-105.813,173.712,35.980,156.751
C04434=1059.696,335.514,-105.848,173.716,35.984,156.752
C04435=1059.703,335.762,-105.883,173.720,35.990,156.753
C04436=1059.709,336.009,-105.918,173.724,35.994,156.754
C04437=1059.716,336.257,-105.953,173.727,35.999,156.755
C04438=1059.724,336.505,-105.989,173.732,36.003,156.756
C04439=1059.730,336.752,-106.024,173.736,36.008,156.757
C04440=1059.737,336.999,-106.059,173.739,36.013,156.759
C04441=1059.743,337.247,-106.095,173.744,36.018,156.760
C04442=1059.750,337.494,-106.130,173.747,36.022,156.761
C04443=1059.757,337.742,-106.165,173.751,36.027,156.762
C04444=1059.763,337.989,-106.201,173.754,36.032,156.763
C04445=1059.769,338.237,-106.236,173.759,36.036,156.764
C04446=1059.777,338.484,-106.272,173.762,36.042,156.765
C04447=1059.783,338.731,-106.307,173.766,36.046,156.766
C04448=1059.789,338.979,-106.342,173.771,36.051,156.767
C04449=1059.796,339.226,-106.378,173.774,36.056,156.768
C04450=1059.802,339.474,-106.413,173.778,36.060,156.769
C04451=1059.810,339.721,-106.450,173.782,36.065,156.770
C04452=1059.817,339.968,-106.485,173.786,36.070,156.771
C04453=1059.823,340.216,-106.520,173.790,36.075,156.772
C04454=1059.830,340.463,-106.556,173.794,36.080,156.773
C04455=1059.836,340.710,-106.591,173.798,36.085,156.775
C04456=1059.843,340.958,-106.627,173.802,36.089,156.776
C04457=1059.850,341.205,-106.663,173.806,36.094,156.777
C04458=1059.857,341.453,-106.698,173.809,36.099,156.778
C04459=1059.863,341.700,-106.735,173.814,36.104,156.779
C04460=1059.870,341.947,-106.770,173.818,36.109,156.780
C04461=1059.877,342.194,-106.806,173.822,36.114,156.781
C04462=1059.884,342.442,-106.842,173.826,36.118,156.782
C04463=1059.891,342.689,-106.878,173.829,36.123,156.783
C04464=1059.897,342.937,-106.914,173.834,36.128,156.784
C04465=1059.904,343.183,-106.949,173.837,36.133,156.786
C04466=1059.911,343.432,-106.985,173.842,36.138,156.787
C04467=1059.918,343.679,-107.021,173.846,36.143,156.788
C04468=1059.924,343.926,-107.057,173.850,36.148,156.789
C04469=1059.931,344.173,-107.093,173.854,36.153,156.790
C04470=1059.938,344.421,-107.130,173.858,36.158,156.791
C04471=1059.944,344.668,-107.165,173.862,36.163,156.792
C04472=1059.951,344.915,-107.201,173.866,36.168,156.793
C04473=1059.958,345.163,-107.238,173.870,36.173,156.794
C04474=1059.964,345.407,-107.273,173.874,36.178,156.796
C04475=1059.971,345.650,-107.309,173.879,36.182,156.797
C04476=1059.977,345.895,-107.345,173.882,36.187,156.798
C04477=1059.984,346.139,-107.380,173.886,36.193,156.799
C04478=1059.991,346.383,-107.417,173.890,36.198,156.800
C04479=1059.998,346.628,-107.452,173.894,36.202,156.801
C04480=1060.004,346.871,-107.487,173.899,36.207,156.802
C04481=1060.011,347.116,-107.523,173.902,36.212,156.803
C04482=1060.018,347.363,-107.560,173.907,36.217,156.805
C04483=1060.025,347.610,-107.596,173.911,36.222,156.806
C04484=1060.031,347.857,-107.632,173.914,36.228,156.807
C04485=1060.038,348.105,-107.669,173.919,36.233,156.808
C04486=1060.045,348.352,-107.705,173.922,36.238,156.809
C04487=1060.052,348.599,-107.742,173.927,36.243,156.810
C04488=1060.058,348.846,-107.778,173.932,36.248,156.812
C04489=1060.065,349.094,-107.815,173.935,36.253,156.813
C04490=1060.072,349.341,-107.851,173.940,36.258,156.814
C04491=1060.079,349.587,-107.888,173.944,36.263,156.815
C04492=1060.086,349.835,-107.925,173.948,36.268,156.816
C04493=1060.093,350.082,-107.961,173.952,36.273,156.817
C04494=1060.100,350.330,-107.998,173.957,36.278,156.819
C04495=1060.106,350.577,-108.034,173.960,36.283,156.820
C04496=1060.113,350.824,-108.071,173.965,36.289,156.821
C04497=1060.120,351.071,-108.107,173.969,36.294,156.822
C04498=1060.127,351.318,-108.144,173.973,36.299,156.823
C04499=1060.134,351.565,-108.181,173.977,36.304,156.825
C04500=1060.141,351.813,-108.217,173.982,36.309,156.826
C04501=1060.148,352.060,-108.255,173.986,36.315,156.827
C04502=1060.154,352.307,-108.291,173.990,36.320,156.828
C04503=1060.161,352.555,-108.328,173.995,36.325,156.829
C04504=1060.168,352.801,-108.365,173.998,36.331,156.831
C04505=1060.175,353.049,-108.402,174.003,36.336,156.832
C04506=1060.181,353.296,-108.439,174.007,36.341,156.833
C04507=1060.188,353.543,-108.476,174.012,36.346,156.834
C04508=1060.195,353.790,-108.513,174.016,36.352,156.835
C04509=1060.202,354.038,-108.550,174.020,36.357,156.837
C04510=1060.209,354.285,-108.588,174.025,36.362,156.838
C04511=1060.216,354.532,-108.624,174.028,36.368,156.839
C04512=1060.223,354.779,-108.662,174.033,36.373,156.840
C04513=1060.229,355.026,-108.698,174.038,36.378,156.842
C04514=1060.236,355.273,-108.736,174.041,36.384,156.843
C04515=1060.243,355.521,-108.772,174.046,36.389,156.844
C04516=1060.250,355.767,-108.810,174.051,36.394,156.845
C04517=1060.257,356.014,-108.847,174.055,36.400,156.847
C04518=1060.264,356.262,-108.884,174.059,36.405,156.848
C04519=1060.271,356.509,-108.921,174.063,36.410,156.849
C04520=1060.278,356.756,-108.959,174.068,36.416,156.850
C04521=1060.285,357.003,-108.996,174.072,36.421,156.851
C04522=1060.292,357.251,-109.033,174.076,36.427,156.853
C04523=1060.299,357.497,-109.070,174.081,36.432,156.854
C04524=1060.306,357.744,-109.108,174.086,36.437,156.855
C04525=1060.313,357.991,-109.145,174.090,36.443,156.857
C04526=1060.321,358.238,-109.183,174.094,36.449,156.858
C04527=1060.327,358.486,-109.219,174.099,36.454,156.859
C04528=1060.334,358.733,-109.257,174.104,36.459,156.860
C04529=1060.341,358.980,-109.295,174.107,36.465,156.862
C04530=1060.348,359.226,-109.333,174.112,36.470,156.863
C04531=1060.354,359.472,-109.370,174.117,36.476,156.864
C04532=1060.362,359.718,-109.406,174.121,36.482,156.866
C04533=1060.369,359.965,-109.445,174.126,36.487,156.867
C04534=1060.376,360.211,-109.482,174.130,36.492,156.868
C04535=1060.383,360.457,-109.520,174.134,36.498,156.869
C04536=1060.389,360.704,-109.557,174.139,36.503,156.871
C04537=1060.396,360.949,-109.595,174.144,36.509,156.872
C04538=1060.404,361.197,-109.632,174.148,36.514,156.873
C04539=1060.410,361.444,-109.670,174.152,36.520,156.875
C04540=1060.417,361.691,-109.708,174.157,36.526,156.876
C04541=1060.425,361.938,-109.745,174.162,36.531,156.877
C04542=1060.431,362.185,-109.784,174.166,36.537,156.878
C04543=1060.439,362.432,-109.822,174.170,36.543,156.880
C04544=1060.446,362.679,-109.859,174.175,36.549,156.881
C04545=1060.452,362.927,-109.897,174.180,36.554,156.882
C04546=1060.460,363.173,-109.936,174.185,36.560,156.884
C04547=1060.467,363.420,-109.973,174.189,36.565,156.885
C04548=1060.473,363.667,-110.011,174.193,36.571,156.886
C04549=1060.481,363.914,-110.049,174.198,36.577,156.888
C04550=1060.488,364.161,-110.087,174.203,36.582,156.889
C04551=1060.495,364.408,-110.126,174.208,36.588,156.890
C04552=1060.502,364.655,-110.163,174.212,36.594,156.892
C04553=1060.509,364.902,-110.202,174.216,36.600,156.893
C04554=1060.515,365.149,-110.240,174.221,36.606,156.895
C04555=1060.523,365.396,-110.278,174.226,36.611,156.896
C04556=1060.529,365.643,-110.316,174.231,36.618,156.897
C04557=1060.537,365.890,-110.355,174.236,36.623,156.899
C04558=1060.544,366.136,-110.394,174.240,36.629,156.900
C04559=1060.551,366.384,-110.431,174.244,36.635,156.902
C04560=1060.558,366.630,-110.470,174.249,36.641,156.903
C04561=1060.565,366.877,-110.509,174.254,36.646,156.904
C04562=1060.572,367.124,-110.546,174.259,36.652,156.906
C04563=1060.579,367.371,-110.585,174.264,36.658,156.907
C04564=1060.586,367.618,-110.623,174.268,36.664,156.908
C04565=1060.593,367.864,-110.662,174.273,36.670,156.910
C04566=1060.600,368.112,-110.700,174.277,36.676,156.911
C04567=1060.608,368.359,-110.739,174.282,36.682,156.913
C04568=1060.615,368.606,-110.778,174.287,36.688,156.914
C04569=1060.622,368.852,-110.816,174.292,36.694,156.916
C04570=1060.629,369.099,-110.855,174.297,36.700,156.917
C04571=1060.636,369.346,-110.894,174.302,36.706,156.918
C04572=1060.643,369.593,-110.932,174.307,36.712,156.920
C04573=1060.651,369.840,-110.971,174.311,36.718,156.921
C04574=1060.658,370.087,-111.009,174.315,36.723,156.923
C04575=1060.665,370.333,-111.048,174.320,36.729,156.924
C04576=1060.672,370.580,-111.087,174.325,36.736,156.925
C04577=1060.679,370.827,-111.125,174.330,36.742,156.927
C04578=1060.687,371.074,-111.164,174.335,36.748,156.928
C04579=1060.694,371.321,-111.203,174.340,36.754,156.930
C04580=1060.701,371.568,-111.242,174.345,36.760,156.931
C04581=1060.708,371.815,-111.280,174.350,36.766,156.933
C04582=1060.715,372.062,-111.320,174.355,36.772,156.934
C04583=1060.723,372.308,-111.359,174.360,36.778,156.936
C04584=1060.730,372.555,-111.397,174.365,36.784,156.937
C04585=1060.737,372.802,-111.437,174.370,36.790,156.939
C04586=1060.744,373.066,-111.479,174.375,36.797,156.940
C04587=1060.753,373.329,-111.520,174.380,36.804,156.942
C04588=1060.760,373.593,-111.562,174.386,36.811,156.943
C04589=1060.768,373.857,-111.604,174.391,36.817,156.945
C04590=1060.775,374.103,-111.643,174.396,36.823,156.946
C04591=1060.782,374.351,-111.682,174.401,36.829,156.948
C04592=1060.789,374.597,-111.722,174.406,36.836,156.950
C04593=1060.796,374.844,-111.761,174.411,36.842,156.951
C04594=1060.804,375.091,-111.801,174.416,36.849,156.953
C04595=1060.811,375.337,-111.839,174.420,36.855,156.954
C04596=1060.818,375.584,-111.879,174.426,36.861,156.956
C04597=1060.825,375.831,-111.918,174.430,36.867,156.957
C04598=1060.832,376.077,-111.958,174.435,36.874,156.959
C04599=1060.840,376.324,-111.998,174.440,36.880,156.960
C04600=1060.847,376.571,-112.037,174.445,36.887,156.962
C04601=1060.854,376.817,-112.076,174.450,36.893,156.963
C04602=1060.862,377.064,-112.116,174.455,36.899,156.965
C04603=1060.869,377.310,-112.156,174.460,36.906,156.966
C04604=1060.876,377.558,-112.195,174.465,36.912,156.968
C04605=1060.883,377.804,-112.234,174.471,36.918,156.969
C04606=1060.891,378.051,-112.274,174.477,36.925,156.971
C04607=1060.898,378.297,-112.314,174.482,36.932,156.973
C04608=1060.906,378.544,-112.354,174.487,36.938,156.974
C04609=1060.913,378.791,-112.393,174.492,36.944,156.976
C04610=1060.920,379.038,-112.432,174.497,36.951,156.977
C04611=1060.928,379.284,-112.472,174.502,36.957,156.979
C04612=1060.935,379.531,-112.512,174.507,36.964,156.981
C04613=1060.943,379.778,-112.552,174.513,36.971,156.982
C04614=1060.950,380.024,-112.591,174.518,36.977,156.984
C04615=1060.958,380.271,-112.631,174.523,36.984,156.985
C04616=1060.966,380.518,-112.671,174.528,36.990,156.987
C04617=1060.972,380.764,-112.711,174.533,36.997,156.989
C04618=1060.980,381.011,-112.751,174.538,37.003,156.990
C04619=1060.987,381.257,-112.792,174.543,37.010,156.992
C04620=1060.994,381.504,-112.832,174.549,37.017,156.993
C04621=1061.002,381.751,-112.872,174.554,37.024,156.995
C04622=1061.009,381.997,-112.912,174.559,37.030,156.997
C04623=1061.016,382.244,-112.953,174.565,37.037,156.998
C04624=1061.024,382.491,-112.993,174.570,37.044,157.000
C04625=1061.031,382.737,-113.032,174.576,37.050,157.002
C04626=1061.038,382.984,-113.074,174.581,37.057,157.003
C04627=1061.046,383.230,-113.113,174.586,37.064,157.005
C04628=1061.053,383.477,-113.153,174.591,37.071,157.007
C04629=1061.060,383.723,-113.194,174.596,37.078,157.008
C04630=1061.068,383.970,-113.234,174.602,37.084,157.010
C04631=1061.075,384.216,-113.275,174.608,37.091,157.012
C04632=1061.083,384.463,-113.315,174.613,37.098,157.013
C04633=1061.091,384.709,-113.356,174.618,37.105,157.015
C04634=1061.098,384.956,-113.396,174.624,37.112,157.017
C04635=1061.106,385.203,-113.437,174.629,37.119,157.018
C04636=1061.112,385.449,-113.478,174.634,37.126,157.020
C04637=1061.120,385.696,-113.517,174.641,37.133,157.022
C04638=1061.128,385.942,-113.558,174.646,37.140,157.024
C04639=1061.135,386.188,-113.599,174.651,37.146,157.025
C04640=1061.143,386.435,-113.639,174.656,37.153,157.027
C04641=1061.150,386.682,-113.680,174.662,37.161,157.029
C04642=1061.160,386.976,-113.729,174.669,37.169,157.031
C04643=1061.169,387.271,-113.778,174.675,37.177,157.033
C04644=1061.177,387.566,-113.826,174.681,37.186,157.035
C04645=1061.187,387.860,-113.875,174.688,37.194,157.037
C04646=1061.195,388.107,-113.916,174.694,37.201,157.039
C04647=1061.202,388.353,-113.957,174.699,37.208,157.041
C04648=1061.210,388.600,-113.998,174.706,37.215,157.042
C04649=1061.217,388.846,-114.039,174.711,37.222,157.044
C04650=1061.225,389.092,-114.080,174.716,37.229,157.046
C04651=1061.233,389.339,-114.121,174.722,37.237,157.048
C04652=1061.241,389.585,-114.161,174.728,37.244,157.050
C04653=1061.248,389.832,-114.203,174.734,37.251,157.051
C04654=1061.256,390.078,-114.243,174.739,37.258,157.053
C04655=1061.263,390.325,-114.285,174.744,37.266,157.055
C04656=1061.271,390.571,-114.326,174.751,37.273,157.057
C04657=1061.279,390.817,-114.367,174.756,37.280,157.059
C04658=1061.286,391.064,-114.408,174.762,37.287,157.060
C04659=1061.293,391.310,-114.450,174.768,37.295,157.062
C04660=1061.302,391.556,-114.491,174.774,37.302,157.064
C04661=1061.310,391.803,-114.532,174.779,37.310,157.066
C04662=1061.317,392.050,-114.574,174.784,37.317,157.068
C04663=1061.325,392.296,-114.616,174.791,37.324,157.070
C04664=1061.333,392.542,-114.656,174.796,37.332,157.071
C04665=1061.340,392.788,-114.698,174.802,37.339,157.073
C04666=1061.348,393.035,-114.739,174.808,37.347,157.075
C04667=1061.355,393.281,-114.781,174.814,37.354,157.077
C04668=1061.364,393.528,-114.822,174.819,37.361,157.079
C04669=1061.371,393.774,-114.864,174.826,37.369,157.081
C04670=1061.379,394.020,-114.906,174.831,37.377,157.083
C04671=1061.386,394.266,-114.948,174.837,37.384,157.085
C04672=1061.394,394.512,-114.989,174.843,37.392,157.087
C04673=1061.402,394.759,-115.031,174.849,37.399,157.088
C04674=1061.409,395.005,-115.073,174.856,37.407,157.090
C04675=1061.417,395.251,-115.115,174.861,37.415,157.092
C04676=1061.425,395.498,-115.157,174.867,37.422,157.094
C04677=1061.433,395.744,-115.199,174.873,37.430,157.096
C04678=1061.441,395.990,-115.240,174.879,37.437,157.098
C04679=1061.448,396.236,-115.282,174.885,37.446,157.100
C04680=1061.456,396.483,-115.324,174.891,37.453,157.102
C04681=1061.464,396.729,-115.366,174.897,37.461,157.104
C04682=1061.472,396.976,-115.408,174.903,37.469,157.106
C04683=1061.480,397.222,-115.450,174.909,37.476,157.108
C04684=1061.488,397.468,-115.493,174.915,37.484,157.110
C04685=1061.496,397.714,-115.535,174.921,37.492,157.112
C04686=1061.503,397.960,-115.577,174.928,37.500,157.114
C04687=1061.511,398.207,-115.619,174.933,37.508,157.116
C04688=1061.518,398.453,-115.661,174.940,37.515,157.118
C04689=1061.527,398.699,-115.704,174.945,37.523,157.120
C04690=1061.534,398.945,-115.746,174.952,37.531,157.122
C04691=1061.543,399.192,-115.789,174.958,37.539,157.124
C04692=1061.550,399.438,-115.831,174.964,37.548,157.126
C04693=1061.559,399.684,-115.874,174.970,37.556,157.128
C04694=1061.566,399.930,-115.916,174.977,37.564,157.130
C04695=1061.574,400.177,-115.958,174.983,37.571,157.132
C04696=1061.582,400.422,-116.001,174.989,37.580,157.134
C04697=1061.590,400.669,-116.043,174.995,37.588,157.136
C04698=1061.600,400.981,-116.097,175.003,37.598,157.139
C04699=1061.610,401.292,-116.151,175.011,37.608,157.142
C04700=1061.620,401.604,-116.205,175.019,37.618,157.144
C04701=1061.631,401.915,-116.260,175.027,37.629,157.147
C04702=1061.638,402.162,-116.303,175.034,37.637,157.149
C04703=1061.646,402.408,-116.345,175.040,37.645,157.151
C04704=1061.655,402.654,-116.388,175.046,37.653,157.153
C04705=1061.663,402.900,-116.431,175.052,37.661,157.155
C04706=1061.670,403.146,-116.474,175.059,37.670,157.158
C04707=1061.678,403.392,-116.517,175.066,37.678,157.160
C04708=1061.686,403.639,-116.560,175.071,37.687,157.162
C04709=1061.694,403.885,-116.603,175.078,37.695,157.164
C04710=1061.703,404.131,-116.646,175.085,37.703,157.166
C04711=1061.710,404.377,-116.689,175.091,37.712,157.168
C04712=1061.719,404.623,-116.732,175.098,37.720,157.170
C04713=1061.726,404.869,-116.776,175.105,37.729,157.173
C04714=1061.735,405.115,-116.819,175.111,37.737,157.175
C04715=1061.743,405.362,-116.862,175.117,37.746,157.177
C04716=1061.751,405.608,-116.905,175.124,37.754,157.179
C04717=1061.759,405.854,-116.949,175.130,37.763,157.182
C04718=1061.767,406.100,-116.992,175.137,37.771,157.184
C04719=1061.774,406.346,-117.035,175.144,37.780,157.186
C04720=1061.782,406.592,-117.079,175.150,37.788,157.188
C04721=1061.791,406.838,-117.123,175.157,37.797,157.191
C04722=1061.799,407.084,-117.166,175.164,37.806,157.193
C04723=1061.807,407.330,-117.209,175.171,37.815,157.195
C04724=1061.815,407.576,-117.254,175.177,37.823,157.197
C04725=1061.823,407.822,-117.297,175.184,37.832,157.200
C04726=1061.832,408.068,-117.340,175.191,37.841,157.202
C04727=1061.840,408.314,-117.385,175.198,37.850,157.204
C04728=1061.847,408.560,-117.428,175.205,37.858,157.206
C04729=1061.856,408.806,-117.472,175.211,37.867,157.209
C04730=1061.864,409.052,-117.516,175.218,37.876,157.211
C04731=1061.873,409.299,-117.560,175.225,37.885,157.213
C04732=1061.881,409.545,-117.603,175.232,37.894,157.216
C04733=1061.889,409.790,-117.648,175.239,37.903,157.218
C04734=1061.897,410.036,-117.692,175.246,37.912,157.221
C04735=1061.905,410.283,-117.736,175.252,37.921,157.223
C04736=1061.914,410.528,-117.779,175.259,37.930,157.225
C04737=1061.922,410.774,-117.824,175.266,37.939,157.228
C04738=1061.931,411.020,-117.868,175.273,37.948,157.230
C04739=1061.939,411.266,-117.911,175.281,37.957,157.232
C04740=1061.947,411.512,-117.956,175.288,37.966,157.235
C04741=1061.956,411.758,-118.000,175.295,37.975,157.237
C04742=1061.964,412.004,-118.045,175.302,37.984,157.240
C04743=1061.973,412.250,-118.089,175.308,37.993,157.242
C04744=1061.981,412.495,-118.133,175.315,38.002,157.244
C04745=1061.990,412.742,-118.178,175.323,38.011,157.247
C04746=1061.998,412.988,-118.222,175.330,38.021,157.249
C04747=1062.007,413.234,-118.266,175.337,38.030,157.252
C04748=1062.015,413.479,-118.310,175.344,38.039,157.254
C04749=1062.023,413.725,-118.355,175.352,38.048,157.257
C04750=1062.032,413.972,-118.399,175.359,38.058,157.259
C04751=1062.040,414.217,-118.444,175.366,38.067,157.262
C04752=1062.049,414.463,-118.489,175.373,38.077,157.264
C04753=1062.057,414.709,-118.533,175.381,38.086,157.267
C04754=1062.068,415.025,-118.591,175.390,38.098,157.270
C04755=1062.079,415.343,-118.650,175.400,38.111,157.273
C04756=1062.090,415.659,-118.707,175.409,38.123,157.277
C04757=1062.101,415.976,-118.765,175.419,38.135,157.280
C04758=1062.109,416.221,-118.810,175.426,38.145,157.282
C04759=1062.118,416.467,-118.854,175.434,38.154,157.285
C04760=1062.126,416.714,-118.901,175.441,38.164,157.288
C04761=1062.134,416.959,-118.945,175.449,38.174,157.290
C04762=1062.143,417.205,-118.990,175.457,38.184,157.293
C04763=1062.152,417.450,-119.035,175.464,38.193,157.295
C04764=1062.161,417.696,-119.081,175.472,38.203,157.298
C04765=1062.169,417.943,-119.125,175.479,38.213,157.301
C04766=1062.178,418.188,-119.170,175.487,38.223,157.303
C04767=1062.187,418.434,-119.216,175.494,38.232,157.306
C04768=1062.196,418.679,-119.261,175.503,38.242,157.309
C04769=1062.203,418.925,-119.307,175.510,38.252,157.311
C04770=1062.212,419.171,-119.352,175.518,38.262,157.314
C04771=1062.221,419.416,-119.398,175.525,38.272,157.317
C04772=1062.230,419.662,-119.443,175.533,38.282,157.319
C04773=1062.239,419.908,-119.489,175.541,38.292,157.322
C04774=1062.248,420.153,-119.534,175.549,38.302,157.325
C04775=1062.256,420.399,-119.580,175.556,38.312,157.328
C04776=1062.265,420.645,-119.626,175.565,38.323,157.330
C04777=1062.274,420.890,-119.671,175.573,38.332,157.333
C04778=1062.282,421.137,-119.717,175.580,38.343,157.336
C04779=1062.292,421.382,-119.763,175.589,38.353,157.339
C04780=1062.299,421.627,-119.809,175.597,38.363,157.342
C04781=1062.309,421.872,-119.855,175.604,38.374,157.344
C04782=1062.318,422.118,-119.901,175.613,38.384,157.347
C04783=1062.326,422.364,-119.947,175.620,38.394,157.350
C04784=1062.335,422.609,-119.993,175.629,38.405,157.353
C04785=1062.344,422.855,-120.039,175.637,38.415,157.356
C04786=1062.353,423.101,-120.085,175.645,38.426,157.359
C04787=1062.361,423.346,-120.132,175.653,38.436,157.361
C04788=1062.370,423.592,-120.178,175.661,38.446,157.364
C04789=1062.379,423.837,-120.223,175.670,38.457,157.367
C04790=1062.388,424.083,-120.270,175.678,38.468,157.370
C04791=1062.397,424.328,-120.316,175.686,38.478,157.373
C04792=1062.406,424.574,-120.363,175.694,38.488,157.376
C04793=1062.416,424.820,-120.409,175.703,38.499,157.379
C04794=1062.424,425.065,-120.456,175.711,38.510,157.382
C04795=1062.434,425.310,-120.502,175.720,38.520,157.385
C04796=1062.442,425.556,-120.549,175.728,38.531,157.388
C04797=1062.451,425.801,-120.595,175.737,38.542,157.391
C04798=1062.460,426.047,-120.642,175.744,38.553,157.394
C04799=1062.470,426.292,-120.688,175.753,38.563,157.397
C04800=1062.478,426.538,-120.735,175.762,38.574,157.400
C04801=1062.487,426.783,-120.782,175.770,38.585,157.403
C04802=1062.497,427.029,-120.829,175.779,38.596,157.406
C04803=1062.506,427.274,-120.876,175.787,38.607,157.409
C04804=1062.514,427.520,-120.922,175.796,38.618,157.412
C04805=1062.524,427.765,-120.970,175.805,38.629,157.415
C04806=1062.533,428.011,-121.016,175.814,38.640,157.418
C04807=1062.542,428.255,-121.064,175.822,38.651,157.421
C04808=1062.551,428.502,-121.111,175.831,38.663,157.424
C04809=1062.560,428.746,-121.158,175.840,38.673,157.427
C04810=1062.569,428.976,-121.202,175.848,38.684,157.430
C04811=1062.577,429.206,-121.247,175.857,38.695,157.433
C04812=1062.587,429.437,-121.291,175.865,38.705,157.436
C04813=1062.595,429.667,-121.335,175.873,38.716,157.439
C04814=1062.603,429.897,-121.380,175.882,38.726,157.442
C04815=1062.613,430.127,-121.424,175.890,38.737,157.445
C04816=1062.621,430.357,-121.469,175.898,38.748,157.448
C04817=1062.629,430.587,-121.513,175.907,38.758,157.451
C04818=1062.639,430.833,-121.561,175.916,38.770,157.454
C04819=1062.648,431.079,-121.609,175.925,38.781,157.458
C04820=1062.657,431.324,-121.656,175.934,38.793,157.461
C04821=1062.666,431.569,-121.704,175.943,38.804,157.464
C04822=1062.676,431.813,-121.752,175.952,38.816,157.467
C04823=1062.685,432.059,-121.800,175.961,38.828,157.471
C04824=1062.694,432.305,-121.848,175.971,38.840,157.474
C04825=1062.703,432.549,-121.895,175.980,38.851,157.477
C04826=1062.713,432.794,-121.944,175.989,38.863,157.481
C04827=1062.723,433.040,-121.992,175.999,38.875,157.484
C04828=1062.731,433.285,-122.039,176.008,38.887,157.487
C04829=1062.741,433.530,-122.088,176.017,38.898,157.491
C04830=1062.751,433.775,-122.136,176.027,38.911,157.494
C04831=1062.760,434.020,-122.184,176.036,38.922,157.498
C04832=1062.769,434.265,-122.232,176.047,38.934,157.501
C04833=1062.779,434.510,-122.280,176.056,38.946,157.504
C04834=1062.789,434.755,-122.328,176.065,38.958,157.508
C04835=1062.798,435.000,-122.377,176.075,38.971,157.511
C04836=1062.808,435.245,-122.425,176.084,38.982,157.515
C04837=1062.818,435.491,-122.473,176.094,38.994,157.518
C04838=1062.827,435.736,-122.522,176.104,39.007,157.522
C04839=1062.837,435.981,-122.570,176.114,39.019,157.525
C04840=1062.846,436.226,-122.619,176.124,39.031,157.529
C04841=1062.856,436.471,-122.668,176.133,39.044,157.532
C04842=1062.866,436.716,-122.716,176.144,39.056,157.536
C04843=1062.875,436.961,-122.765,176.153,39.068,157.539
C04844=1062.886,437.205,-122.814,176.163,39.081,157.543
C04845=1062.895,437.450,-122.863,176.173,39.093,157.547
C04846=1062.905,437.695,-122.911,176.183,39.106,157.550
C04847=1062.914,437.941,-122.960,176.193,39.118,157.554
C04848=1062.924,438.185,-123.010,176.204,39.131,157.558
C04849=1062.935,438.431,-123.059,176.213,39.143,157.561
C04850=1062.949,438.797,-123.132,176.229,39.162,157.567
C04851=1062.963,439.164,-123.206,176.244,39.181,157.572
C04852=1062.978,439.531,-123.280,176.260,39.200,157.578
C04853=1062.993,439.897,-123.353,176.275,39.220,157.584
C04854=1063.003,440.143,-123.403,176.286,39.233,157.587
C04855=1063.013,440.387,-123.452,176.296,39.246,157.591
C04856=1063.022,440.632,-123.502,176.307,39.258,157.595
C04857=1063.033,440.877,-123.552,176.317,39.271,157.599
C04858=1063.042,441.122,-123.601,176.328,39.285,157.603
C04859=1063.053,441.367,-123.651,176.338,39.298,157.606
C04860=1063.062,441.611,-123.701,176.348,39.311,157.610
C04861=1063.072,441.856,-123.750,176.359,39.324,157.614
C04862=1063.083,442.100,-123.801,176.370,39.337,157.618
C04863=1063.093,442.345,-123.850,176.381,39.351,157.622
C04864=1063.103,442.590,-123.901,176.392,39.364,157.626
C04865=1063.113,442.835,-123.950,176.403,39.377,157.630
C04866=1063.126,443.128,-124.010,176.416,39.393,157.635
C04867=1063.137,443.421,-124.071,176.429,39.410,157.640
C04868=1063.150,443.714,-124.131,176.442,39.426,157.644
C04869=1063.161,444.008,-124.191,176.456,39.442,157.649
C04870=1063.172,444.253,-124.242,176.466,39.456,157.653
C04871=1063.182,444.497,-124.292,176.477,39.469,157.657
C04872=1063.192,444.742,-124.342,176.489,39.483,157.662
C04873=1063.202,444.987,-124.393,176.500,39.497,157.666
C04874=1063.213,445.231,-124.443,176.511,39.511,157.670
C04875=1063.223,445.475,-124.494,176.522,39.525,157.674
C04876=1063.233,445.720,-124.545,176.535,39.539,157.678
C04877=1063.244,445.964,-124.595,176.546,39.553,157.682
C04878=1063.254,446.209,-124.646,176.558,39.566,157.686
C04879=1063.264,446.454,-124.697,176.569,39.580,157.691
C04880=1063.276,446.698,-124.748,176.580,39.595,157.695
C04881=1063.286,446.942,-124.799,176.592,39.609,157.699
C04882=1063.297,447.186,-124.849,176.604,39.623,157.704
C04883=1063.306,447.430,-124.900,176.616,39.637,157.708
C04884=1063.318,447.673,-124.951,176.627,39.651,157.712
C04885=1063.329,447.917,-125.001,176.639,39.665,157.716
C04886=1063.342,448.161,-125.050,176.651,39.678,157.720
C04887=1063.356,448.405,-125.098,176.663,39.692,157.724
C04888=1063.371,448.650,-125.147,176.675,39.705,157.728
C04889=1063.387,448.895,-125.194,176.687,39.718,157.732
C04890=1063.403,449.139,-125.241,176.700,39.730,157.736
C04891=1063.421,449.385,-125.287,176.712,39.742,157.740
C04892=1063.440,449.630,-125.333,176.724,39.754,157.744
C04893=1063.460,449.876,-125.378,176.736,39.766,157.747
C04894=1063.123,449.883,-125.648,176.729,39.886,157.780
C04895=1063.104,449.638,-125.603,176.717,39.875,157.777
C04896=1063.084,449.392,-125.558,176.705,39.863,157.773
C04897=1063.067,449.147,-125.511,176.692,39.851,157.769
C04898=1063.050,448.903,-125.465,176.680,39.839,157.765
C04899=1063.034,448.658,-125.418,176.667,39.826,157.761
C04900=1063.019,448.413,-125.370,176.655,39.813,157.757
C04901=1063.006,448.168,-125.321,176.643,39.800,157.753
C04902=1062.992,447.925,-125.272,176.631,39.786,157.749
C04903=1062.980,447.681,-125.222,176.618,39.773,157.745
C04904=1062.969,447.436,-125.171,176.607,39.759,157.741
C04905=1062.958,447.193,-125.121,176.595,39.744,157.736
C04906=1062.947,446.950,-125.070,176.584,39.730,157.732
C04907=1062.937,446.705,-125.019,176.571,39.717,157.728
C04908=1062.927,446.461,-124.967,176.560,39.702,157.723
C04909=1062.916,446.217,-124.917,176.548,39.688,157.719
C04910=1062.905,445.972,-124.866,176.537,39.674,157.715
C04911=1062.895,445.727,-124.815,176.526,39.660,157.711
C04912=1062.886,445.483,-124.765,176.513,39.647,157.707
C04913=1062.875,445.239,-124.714,176.502,39.633,157.702
C04914=1062.864,444.994,-124.663,176.491,39.619,157.698
C04915=1062.854,444.749,-124.613,176.479,39.605,157.694
C04916=1062.843,444.505,-124.562,176.468,39.592,157.690
C04917=1062.833,444.261,-124.512,176.457,39.578,157.686
C04918=1062.824,444.015,-124.461,176.445,39.564,157.682
C04919=1062.811,443.741,-124.405,176.433,39.549,157.677
C04920=1062.801,443.468,-124.349,176.420,39.534,157.673
C04921=1062.788,443.194,-124.292,176.408,39.519,157.668
C04922=1062.778,442.920,-124.236,176.395,39.504,157.664
C04923=1062.767,442.675,-124.186,176.385,39.490,157.660
C04924=1062.758,442.430,-124.137,176.374,39.477,157.656
C04925=1062.747,442.186,-124.086,176.363,39.464,157.652
C04926=1062.737,441.940,-124.036,176.352,39.451,157.648
C04927=1062.727,441.696,-123.987,176.341,39.438,157.644
C04928=1062.717,441.451,-123.937,176.331,39.424,157.640
C04929=1062.707,441.206,-123.887,176.320,39.411,157.636
C04930=1062.697,440.962,-123.837,176.309,39.398,157.632
C04931=1062.686,440.717,-123.787,176.298,39.385,157.629
C04932=1062.677,440.473,-123.737,176.288,39.373,157.625
C04933=1062.667,440.227,-123.688,176.277,39.359,157.621
C04934=1062.657,439.982,-123.639,176.266,39.346,157.617
C04935=1062.647,439.738,-123.589,176.257,39.334,157.613
C04936=1062.637,439.493,-123.540,176.246,39.321,157.610
C04937=1062.627,439.248,-123.490,176.236,39.308,157.606
C04938=1062.617,439.003,-123.441,176.225,39.296,157.602
C04939=1062.607,438.759,-123.392,176.215,39.283,157.599
C04940=1062.598,438.513,-123.343,176.204,39.270,157.595
C04941=1062.588,438.269,-123.293,176.195,39.258,157.591
C04942=1062.578,438.024,-123.245,176.184,39.245,157.587
C04943=1062.569,437.779,-123.195,176.174,39.232,157.584
C04944=1062.559,437.534,-123.147,176.164,39.220,157.580
C04945=1062.548,437.288,-123.098,176.154,39.208,157.577
C04946=1062.538,437.044,-123.048,176.144,39.195,157.573
C04947=1062.529,436.799,-123.000,176.134,39.183,157.569
C04948=1062.519,436.554,-122.951,176.124,39.171,157.566
C04949=1062.509,436.309,-122.903,176.114,39.158,157.562
C04950=1062.499,436.064,-122.854,176.104,39.146,157.559
C04951=1062.490,435.819,-122.805,176.094,39.134,157.555
C04952=1062.481,435.574,-122.757,176.085,39.122,157.552
C04953=1062.471,435.329,-122.708,176.074,39.109,157.548
C04954=1062.461,435.084,-122.660,176.065,39.098,157.545
C04955=1062.451,434.839,-122.611,176.055,39.086,157.541
C04956=1062.442,434.593,-122.563,176.046,39.073,157.538
C04957=1062.432,434.348,-122.515,176.036,39.062,157.534
C04958=1062.422,434.103,-122.466,176.026,39.049,157.531
C04959=1062.413,433.858,-122.419,176.016,39.038,157.527
C04960=1062.404,433.613,-122.370,176.007,39.025,157.524
C04961=1062.394,433.369,-122.322,175.998,39.014,157.521
C04962=1062.384,433.123,-122.274,175.988,39.002,157.517
C04963=1062.375,432.878,-122.225,175.979,38.990,157.514
C04964=1062.366,432.633,-122.178,175.969,38.979,157.511
C04965=1062.356,432.387,-122.130,175.960,38.967,157.507
C04966=1062.347,432.142,-122.082,175.951,38.955,157.504
C04967=1062.338,431.898,-122.034,175.942,38.943,157.500
C04968=1062.328,431.652,-121.986,175.932,38.932,157.497
C04969=1062.320,431.407,-121.939,175.923,38.920,157.494
C04970=1062.310,431.162,-121.890,175.914,38.909,157.491
C04971=1062.298,430.841,-121.828,175.902,38.894,157.486
C04972=1062.286,430.520,-121.766,175.890,38.879,157.482
C04973=1062.274,430.198,-121.703,175.877,38.864,157.478
C04974=1062.261,429.877,-121.641,175.865,38.849,157.474
C04975=1062.251,429.614,-121.591,175.856,38.837,157.470
C04976=1062.241,429.350,-121.540,175.846,38.825,157.467
C04977=1062.231,429.087,-121.489,175.837,38.813,157.463
C04978=1062.222,428.825,-121.438,175.827,38.801,157.460
C04979=1062.213,428.579,-121.391,175.818,38.790,157.457
C04980=1062.203,428.334,-121.344,175.810,38.779,157.454
C04981=1062.194,428.089,-121.296,175.801,38.768,157.451
C04982=1062.185,427.843,-121.250,175.792,38.757,157.448
C04983=1062.176,427.598,-121.202,175.783,38.745,157.445
C04984=1062.166,427.352,-121.156,175.775,38.735,157.442
C04985=1062.158,427.107,-121.109,175.766,38.724,157.439
C04986=1062.149,426.862,-121.062,175.757,38.712,157.435
C04987=1062.139,426.616,-121.015,175.749,38.702,157.432
C04988=1062.131,426.370,-120.968,175.740,38.691,157.429
C04989=1062.121,426.126,-120.921,175.731,38.680,157.426
C04990=1062.112,425.880,-120.874,175.723,38.670,157.423
C04991=1062.103,425.634,-120.828,175.714,38.659,157.420
C04992=1062.094,425.389,-120.781,175.706,38.648,157.417
C04993=1062.085,425.144,-120.735,175.698,38.638,157.414
C04994=1062.076,424.898,-120.689,175.689,38.627,157.411
C04995=1062.066,424.652,-120.642,175.681,38.616,157.408
C04996=1062.058,424.407,-120.595,175.672,38.606,157.406
C04997=1062.048,424.162,-120.549,175.664,38.595,157.403
C04998=1062.040,423.916,-120.503,175.656,38.584,157.400
C04999=1062.031,423.670,-120.457,175.648,38.574,157.397
C05000=1062.022,423.425,-120.410,175.639,38.564,157.394
C05001=1062.013,423.180,-120.364,175.631,38.553,157.391
C05002=1062.005,422.934,-120.318,175.622,38.543,157.388
C05003=1061.996,422.688,-120.272,175.615,38.533,157.385
C05004=1061.986,422.443,-120.226,175.606,38.522,157.383
C05005=1061.978,422.197,-120.180,175.598,38.512,157.380
C05006=1061.969,421.952,-120.134,175.590,38.501,157.377
C05007=1061.960,421.706,-120.087,175.582,38.491,157.374
C05008=1061.951,421.460,-120.042,175.574,38.481,157.371
C05009=1061.943,421.214,-119.996,175.566,38.471,157.368
C05010=1061.934,420.969,-119.950,175.558,38.460,157.366
C05011=1061.925,420.723,-119.904,175.550,38.451,157.363
C05012=1061.917,420.478,-119.858,175.542,38.440,157.360
C05013=1061.908,420.232,-119.812,175.534,38.430,157.357
C05014=1061.899,419.987,-119.767,175.526,38.420,157.355
C05015=1061.890,419.741,-119.721,175.518,38.410,157.352
C05016=1061.882,419.495,-119.675,175.511,38.401,157.349
C05017=1061.873,419.249,-119.630,175.502,38.390,157.346
C05018=1061.864,419.004,-119.585,175.495,38.380,157.344
C05019=1061.855,418.758,-119.540,175.487,38.371,157.341
C05020=1061.846,418.512,-119.494,175.480,38.361,157.338
C05021=1061.837,418.266,-119.449,175.471,38.351,157.336
C05022=1061.829,418.021,-119.404,175.464,38.341,157.333
C05023=1061.820,417.775,-119.358,175.456,38.331,157.330
C05024=1061.812,417.529,-119.312,175.449,38.322,157.328
C05025=1061.803,417.284,-119.267,175.441,38.312,157.325
C05026=1061.795,417.038,-119.223,175.433,38.302,157.323
C05027=1061.786,416.792,-119.177,175.425,38.292,157.320
C05028=1061.777,416.547,-119.132,175.418,38.283,157.317
C05029=1061.769,416.300,-119.087,175.411,38.273,157.315
C05030=1061.760,416.055,-119.042,175.403,38.264,157.312
C05031=1061.749,415.736,-118.984,175.393,38.251,157.309
C05032=1061.738,415.417,-118.926,175.383,38.239,157.306
C05033=1061.727,415.099,-118.868,175.373,38.226,157.302
C05034=1061.717,414.780,-118.809,175.365,38.214,157.299
C05035=1061.708,414.534,-118.764,175.357,38.205,157.296
C05036=1061.700,414.289,-118.720,175.350,38.195,157.294
C05037=1061.691,414.042,-118.675,175.343,38.186,157.291
C05038=1061.682,413.797,-118.630,175.334,38.177,157.289
C05039=1061.673,413.551,-118.586,175.328,38.168,157.286
C05040=1061.665,413.305,-118.541,175.320,38.158,157.284
C05041=1061.657,413.059,-118.497,175.314,38.149,157.281
C05042=1061.648,412.813,-118.452,175.305,38.140,157.279
C05043=1061.640,412.567,-118.409,175.299,38.131,157.277
C05044=1061.631,412.321,-118.364,175.291,38.121,157.274
C05045=1061.623,412.075,-118.320,175.285,38.112,157.272
C05046=1061.615,411.830,-118.275,175.278,38.103,157.269
C05047=1061.605,411.583,-118.231,175.271,38.094,157.267
C05048=1061.597,411.338,-118.187,175.263,38.085,157.264
C05049=1061.589,411.092,-118.142,175.256,38.076,157.262
C05050=1061.580,410.846,-118.099,175.249,38.067,157.260
C05051=1061.572,410.600,-118.054,175.242,38.058,157.257
C05052=1061.564,410.354,-118.010,175.235,38.049,157.255
C05053=1061.556,410.108,-117.966,175.228,38.040,157.252
C05054=1061.547,409.862,-117.922,175.221,38.031,157.250
C05055=1061.539,409.616,-117.879,175.214,38.022,157.248
C05056=1061.531,409.370,-117.834,175.207,38.013,157.245
C05057=1061.522,409.124,-117.790,175.200,38.005,157.243
C05058=1061.514,408.878,-117.747,175.193,37.996,157.241
C05059=1061.506,408.632,-117.702,175.186,37.987,157.238
C05060=1061.498,408.386,-117.659,175.179,37.978,157.236
C05061=1061.490,408.140,-117.615,175.172,37.969,157.234
C05062=1061.482,407.894,-117.571,175.165,37.961,157.232
C05063=1061.473,407.649,-117.528,175.159,37.952,157.229
C05064=1061.465,407.402,-117.484,175.152,37.943,157.227
C05065=1061.457,407.156,-117.440,175.145,37.934,157.225
C05066=1061.449,406.910,-117.397,175.139,37.926,157.222
C05067=1061.441,406.664,-117.353,175.132,37.917,157.220
C05068=1061.433,406.418,-117.309,175.126,37.908,157.218
C05069=1061.425,406.172,-117.266,175.119,37.900,157.216
C05070=1061.417,405.926,-117.222,175.112,37.891,157.213
C05071=1061.408,405.680,-117.179,175.105,37.883,157.211
C05072=1061.400,405.433,-117.135,175.099,37.874,157.209
C05073=1061.392,405.187,-117.092,175.092,37.866,157.207
C05074=1061.384,404.941,-117.049,175.085,37.857,157.204
C05075=1061.376,404.696,-117.006,175.078,37.849,157.202
C05076=1061.368,404.449,-116.962,175.073,37.840,157.200
C05077=1061.360,404.203,-116.919,175.066,37.832,157.198
C05078=1061.352,403.957,-116.876,175.059,37.824,157.196
C05079=1061.344,403.711,-116.833,175.053,37.815,157.193
C05080=1061.336,403.465,-116.791,175.046,37.807,157.191
C05081=1061.328,403.218,-116.747,175.039,37.799,157.189
C05082=1061.320,402.972,-116.704,175.034,37.791,157.187
C05083=1061.311,402.726,-116.661,175.027,37.782,157.185
C05084=1061.304,402.479,-116.618,175.020,37.774,157.183
C05085=1061.296,402.234,-116.575,175.014,37.766,157.181
C05086=1061.287,401.988,-116.532,175.007,37.758,157.179
C05087=1061.278,401.674,-116.478,174.999,37.748,157.176
C05088=1061.268,401.361,-116.424,174.991,37.737,157.173
C05089=1061.257,401.047,-116.369,174.983,37.727,157.171
C05090=1061.246,400.734,-116.315,174.975,37.717,157.168
C05091=1061.239,400.488,-116.272,174.969,37.709,157.166
C05092=1061.231,400.241,-116.230,174.963,37.701,157.164
C05093=1061.223,399.995,-116.187,174.956,37.693,157.162
C05094=1061.215,399.749,-116.145,174.950,37.684,157.160
C05095=1061.207,399.503,-116.102,174.944,37.676,157.158
C05096=1061.199,399.257,-116.060,174.938,37.668,157.156
C05097=1061.191,399.011,-116.017,174.931,37.660,157.153
C05098=1061.184,398.764,-115.975,174.926,37.652,157.151
C05099=1061.176,398.518,-115.932,174.919,37.645,157.149
C05100=1061.168,398.272,-115.891,174.913,37.637,157.147
C05101=1061.160,398.025,-115.848,174.907,37.629,157.145
C05102=1061.152,397.780,-115.806,174.901,37.621,157.143
C05103=1061.144,397.533,-115.763,174.895,37.613,157.141
C05104=1061.136,397.287,-115.721,174.889,37.605,157.139
C05105=1061.128,397.040,-115.679,174.882,37.598,157.137
C05106=1061.120,396.794,-115.637,174.877,37.590,157.136
C05107=1061.113,396.548,-115.595,174.870,37.582,157.133
C05108=1061.105,396.302,-115.553,174.864,37.575,157.132
C05109=1061.097,396.056,-115.511,174.858,37.567,157.130
C05110=1061.090,395.809,-115.470,174.852,37.559,157.128
C05111=1061.081,395.562,-115.427,174.846,37.551,157.126
C05112=1061.074,395.316,-115.385,174.840,37.544,157.124
C05113=1061.066,395.070,-115.343,174.835,37.536,157.122
C05114=1061.058,394.824,-115.301,174.828,37.529,157.120
C05115=1061.051,394.577,-115.260,174.823,37.521,157.118
C05116=1061.042,394.332,-115.219,174.816,37.514,157.116
C05117=1061.034,394.085,-115.176,174.811,37.506,157.114
C05118=1061.027,393.839,-115.134,174.805,37.499,157.112
C05119=1061.019,393.592,-115.093,174.798,37.491,157.110
C05120=1061.012,393.346,-115.051,174.793,37.484,157.108
C05121=1061.004,393.100,-115.010,174.786,37.476,157.107
C05122=1060.996,392.853,-114.968,174.781,37.469,157.105
C05123=1060.988,392.607,-114.927,174.775,37.461,157.103
C05124=1060.981,392.361,-114.885,174.769,37.454,157.101
C05125=1060.973,392.114,-114.844,174.764,37.446,157.099
C05126=1060.965,391.869,-114.802,174.758,37.439,157.097
C05127=1060.958,391.622,-114.761,174.752,37.432,157.095
C05128=1060.950,391.375,-114.720,174.746,37.424,157.093
C05129=1060.943,391.129,-114.678,174.741,37.417,157.092
C05130=1060.934,390.882,-114.637,174.734,37.410,157.090
C05131=1060.927,390.636,-114.596,174.729,37.403,157.088
C05132=1060.919,390.390,-114.554,174.723,37.395,157.086
C05133=1060.911,390.144,-114.513,174.717,37.388,157.084
C05134=1060.904,389.897,-114.472,174.712,37.381,157.083
C05135=1060.896,389.651,-114.431,174.706,37.373,157.081
C05136=1060.889,389.404,-114.390,174.700,37.366,157.079
C05137=1060.881,389.158,-114.349,174.694,37.359,157.077
C05138=1060.873,388.911,-114.308,174.689,37.352,157.075
C05139=1060.865,388.665,-114.268,174.684,37.345,157.074
C05140=1060.858,388.418,-114.226,174.677,37.338,157.072
C05141=1060.850,388.172,-114.186,174.672,37.331,157.070
C05142=1060.843,387.925,-114.145,174.666,37.324,157.068
C05143=1060.833,387.629,-114.095,174.659,37.315,157.066
C05144=1060.824,387.333,-114.046,174.653,37.307,157.064
C05145=1060.815,387.036,-113.997,174.646,37.299,157.062
C05146=1060.806,386.740,-113.948,174.640,37.290,157.060
C05147=1060.798,386.494,-113.907,174.634,37.283,157.058
C05148=1060.791,386.246,-113.867,174.629,37.276,157.056
C05149=1060.783,386.000,-113.826,174.623,37.269,157.055
C05150=1060.775,385.754,-113.786,174.617,37.262,157.053
C05151=1060.768,385.507,-113.745,174.612,37.256,157.051
C05152=1060.760,385.261,-113.705,174.607,37.249,157.050
C05153=1060.753,385.014,-113.664,174.601,37.242,157.048
C05154=1060.745,384.767,-113.624,174.595,37.235,157.046
C05155=1060.738,384.521,-113.582,174.590,37.228,157.044
C05156=1060.730,384.275,-113.542,174.585,37.221,157.043
C05157=1060.723,384.028,-113.502,174.580,37.214,157.041
C05158=1060.716,383.782,-113.461,174.574,37.207,157.039
C05159=1060.708,383.535,-113.421,174.568,37.201,157.038
C05160=1060.700,383.288,-113.381,174.563,37.194,157.036
C05161=1060.694,383.042,-113.340,174.558,37.187,157.034
C05162=1060.686,382.795,-113.300,174.552,37.181,157.033
C05163=1060.679,382.549,-113.259,174.547,37.173,157.031
C05164=1060.671,382.302,-113.220,174.542,37.167,157.029
C05165=1060.664,382.055,-113.180,174.537,37.160,157.028
C05166=1060.656,381.809,-113.138,174.531,37.153,157.026
C05167=1060.649,381.563,-113.099,174.525,37.147,157.024
C05168=1060.642,381.316,-113.059,174.520,37.140,157.023
C05169=1060.635,381.069,-113.019,174.515,37.134,157.021
C05170=1060.627,380.823,-112.978,174.510,37.126,157.019
C05171=1060.619,380.576,-112.938,174.505,37.120,157.018
C05172=1060.612,380.330,-112.899,174.500,37.113,157.016
C05173=1060.605,380.083,-112.859,174.494,37.107,157.015
C05174=1060.597,379.836,-112.819,174.489,37.101,157.013
C05175=1060.590,379.590,-112.779,174.484,37.094,157.012
C05176=1060.582,379.343,-112.739,174.478,37.088,157.010
C05177=1060.575,379.097,-112.700,174.473,37.081,157.008
C05178=1060.567,378.850,-112.660,174.468,37.074,157.007
C05179=1060.560,378.603,-112.619,174.463,37.068,157.005
C05180=1060.553,378.356,-112.580,174.458,37.062,157.004
C05181=1060.546,378.109,-112.541,174.452,37.055,157.002
C05182=1060.539,377.863,-112.501,174.447,37.049,157.000
C05183=1060.531,377.616,-112.461,174.442,37.042,156.999
C05184=1060.524,377.370,-112.422,174.437,37.036,156.997
C05185=1060.516,377.123,-112.382,174.432,37.030,156.996
C05186=1060.509,376.876,-112.343,174.427,37.023,156.994
C05187=1060.502,376.629,-112.303,174.422,37.017,156.993
C05188=1060.494,376.383,-112.263,174.417,37.010,156.991
C05189=1060.487,376.136,-112.223,174.412,37.004,156.990
C05190=1060.480,375.889,-112.185,174.407,36.998,156.988
C05191=1060.473,375.643,-112.145,174.402,36.992,156.987
C05192=1060.465,375.395,-112.106,174.397,36.985,156.985
C05193=1060.458,375.149,-112.066,174.392,36.979,156.983
C05194=1060.450,374.903,-112.027,174.387,36.972,156.982
C05195=1060.443,374.656,-111.988,174.382,36.966,156.980
C05196=1060.436,374.409,-111.949,174.377,36.960,156.979
C05197=1060.428,374.162,-111.909,174.372,36.954,156.977
C05198=1060.421,373.916,-111.870,174.367,36.948,156.976
C05199=1060.414,373.650,-111.827,174.361,36.941,156.974
C05200=1060.406,373.385,-111.785,174.356,36.934,156.973
C05201=1060.398,373.119,-111.743,174.351,36.927,156.971
C05202=1060.391,372.853,-111.702,174.345,36.921,156.969
C05203=1060.384,372.607,-111.662,174.341,36.915,156.968
C05204=1060.377,372.360,-111.623,174.336,36.909,156.966
C05205=1060.370,372.113,-111.584,174.331,36.902,156.965
C05206=1060.362,371.867,-111.545,174.326,36.896,156.964
C05207=1060.355,371.620,-111.506,174.321,36.890,156.962
C05208=1060.348,371.373,-111.467,174.316,36.884,156.961
C05209=1060.340,371.126,-111.429,174.311,36.878,156.959
C05210=1060.333,370.879,-111.390,174.306,36.872,156.958
C05211=1060.326,370.632,-111.351,174.301,36.866,156.956
C05212=1060.318,370.385,-111.313,174.296,36.860,156.955
C05213=1060.311,370.138,-111.274,174.291,36.854,156.953
C05214=1060.305,369.892,-111.235,174.286,36.848,156.952
C05215=1060.297,369.645,-111.197,174.281,36.842,156.951
C05216=1060.290,369.398,-111.158,174.276,36.836,156.949
C05217=1060.282,369.151,-111.119,174.271,36.830,156.948
C05218=1060.275,368.904,-111.080,174.267,36.825,156.946
C05219=1060.268,368.657,-111.042,174.263,36.819,156.945
C05220=1060.261,368.411,-111.003,174.258,36.812,156.943
C05221=1060.254,368.164,-110.964,174.253,36.807,156.942
C05222=1060.247,367.918,-110.926,174.248,36.801,156.941
C05223=1060.240,367.670,-110.888,174.243,36.795,156.939
C05224=1060.233,367.423,-110.849,174.238,36.789,156.938
C05225=1060.225,367.176,-110.811,174.233,36.783,156.936
C05226=1060.218,366.929,-110.772,174.229,36.777,156.935
C05227=1060.211,366.682,-110.734,174.224,36.771,156.934
C05228=1060.204,366.435,-110.695,174.220,36.765,156.932
C05229=1060.197,366.188,-110.657,174.215,36.760,156.931
C05230=1060.190,365.942,-110.618,174.210,36.754,156.929
C05231=1060.183,365.694,-110.580,174.205,36.748,156.928
C05232=1060.176,365.448,-110.542,174.201,36.742,156.927
C05233=1060.169,365.200,-110.504,174.196,36.737,156.925
C05234=1060.162,364.954,-110.466,174.191,36.731,156.924
C05235=1060.155,364.707,-110.428,174.187,36.725,156.923
C05236=1060.148,364.460,-110.389,174.182,36.719,156.921
C05237=1060.141,364.213,-110.351,174.178,36.713,156.920
C05238=1060.134,363.966,-110.312,174.173,36.708,156.918
C05239=1060.127,363.719,-110.275,174.168,36.702,156.917
C05240=1060.120,363.473,-110.237,174.163,36.697,156.916
C05241=1060.114,363.225,-110.199,174.158,36.690,156.914
C05242=1060.106,362.978,-110.161,174.155,36.685,156.913
C05243=1060.099,362.732,-110.123,174.150,36.679,156.912
C05244=1060.092,362.484,-110.085,174.145,36.674,156.910
C05245=1060.085,362.237,-110.047,174.140,36.668,156.909
C05246=1060.078,361.991,-110.009,174.136,36.663,156.908
C05247=1060.070,361.743,-109.972,174.132,36.657,156.907
C05248=1060.064,361.496,-109.934,174.127,36.651,156.905
C05249=1060.057,361.249,-109.896,174.122,36.646,156.904
C05250=1060.049,361.002,-109.858,174.118,36.640,156.903
C05251=1060.042,360.755,-109.820,174.113,36.635,156.901
C05252=1060.036,360.509,-109.782,174.109,36.629,156.900
C05253=1060.029,360.261,-109.745,174.104,36.624,156.899
C05254=1060.021,360.014,-109.707,174.100,36.618,156.897
C05255=1060.014,359.767,-109.670,174.095,36.612,156.896
C05256=1060.008,359.520,-109.632,174.090,36.607,156.895
C05257=1060.000,359.273,-109.594,174.087,36.601,156.893
C05258=1059.993,359.025,-109.557,174.082,36.596,156.892
C05259=1059.987,358.779,-109.519,174.077,36.591,156.891
C05260=1059.980,358.531,-109.481,174.073,36.585,156.890
C05261=1059.973,358.284,-109.444,174.068,36.579,156.888
C05262=1059.966,358.037,-109.407,174.064,36.574,156.887
C05263=1059.959,357.789,-109.370,174.059,36.569,156.886
C05264=1059.952,357.543,-109.332,174.055,36.563,156.885
C05265=1059.945,357.296,-109.295,174.050,36.558,156.883
C05266=1059.937,357.049,-109.257,174.046,36.553,156.882
C05267=1059.930,356.801,-109.221,174.042,36.547,156.881
C05268=1059.924,356.555,-109.183,174.037,36.542,156.880
C05269=1059.917,356.307,-109.146,174.032,36.536,156.878
C05270=1059.909,356.060,-109.108,174.029,36.531,156.877
C05271=1059.903,355.813,-109.072,174.024,36.526,156.876
C05272=1059.896,355.566,-109.034,174.020,36.520,156.875
C05273=1059.889,355.319,-108.997,174.015,36.515,156.873
C05274=1059.882,355.072,-108.960,174.011,36.509,156.872
C05275=1059.875,354.825,-108.923,174.007,36.504,156.871
C05276=1059.868,354.578,-108.885,174.002,36.499,156.870
C05277=1059.861,354.331,-108.849,173.997,36.494,156.868
C05278=1059.854,354.083,-108.811,173.994,36.489,156.867
C05279=1059.847,353.836,-108.775,173.989,36.483,156.866
C05280=1059.841,353.589,-108.737,173.985,36.478,156.865
C05281=1059.834,353.342,-108.701,173.981,36.472,156.863
C05282=1059.827,353.095,-108.663,173.977,36.467,156.862
C05283=1059.820,352.847,-108.627,173.972,36.462,156.861
C05284=1059.814,352.600,-108.590,173.967,36.457,156.860
C05285=1059.806,352.353,-108.553,173.964,36.452,156.859
C05286=1059.800,352.106,-108.516,173.959,36.447,156.857
C05287=1059.793,351.859,-108.479,173.955,36.441,156.856
C05288=1059.786,351.611,-108.442,173.951,36.436,156.855
C05289=1059.780,351.364,-108.405,173.947,36.431,156.854
C05290=1059.773,351.116,-108.369,173.942,36.426,156.853
C05291=1059.765,350.870,-108.332,173.938,36.421,156.852
C05292=1059.758,350.623,-108.295,173.934,36.415,156.850
C05293=1059.752,350.375,-108.259,173.929,36.410,156.849
C05294=1059.745,350.128,-108.222,173.925,36.405,156.848
C05295=1059.738,349.881,-108.186,173.921,36.400,156.847
C05296=1059.731,349.634,-108.149,173.917,36.395,156.846
C05297=1059.724,349.387,-108.112,173.912,36.390,156.844
C05298=1059.717,349.139,-108.075,173.909,36.385,156.843
C05299=1059.710,348.892,-108.039,173.904,36.380,156.842
C05300=1059.703,348.645,-108.003,173.900,36.375,156.841
C05301=1059.697,348.397,-107.966,173.896,36.370,156.840
C05302=1059.691,348.150,-107.930,173.892,36.364,156.839
C05303=1059.683,347.903,-107.894,173.887,36.359,156.837
C05304=1059.677,347.656,-107.857,173.884,36.354,156.836
C05305=1059.670,347.408,-107.820,173.879,36.349,156.835
C05306=1059.663,347.161,-107.784,173.875,36.344,156.834
C05307=1059.657,346.917,-107.749,173.871,36.339,156.833
C05308=1059.650,346.671,-107.712,173.867,36.335,156.832
C05309=1059.643,346.426,-107.676,173.863,36.329,156.831
C05310=1059.636,346.182,-107.641,173.859,36.324,156.829
C05311=1059.629,345.936,-107.605,173.855,36.319,156.828
C05312=1059.623,345.691,-107.569,173.851,36.315,156.827
C05313=1059.616,345.446,-107.533,173.847,36.310,156.826
C05314=1059.609,345.202,-107.498,173.842,36.305,156.825
C05315=1059.603,344.955,-107.461,173.839,36.299,156.824
C05316=1059.595,344.707,-107.425,173.835,36.295,156.823
C05317=1059.589,344.460,-107.388,173.830,36.290,156.822
C05318=1059.583,344.212,-107.353,173.827,36.285,156.820
C05319=1059.576,343.966,-107.317,173.822,36.280,156.819
C05320=1059.569,343.718,-107.280,173.818,36.275,156.818
C05321=1059.562,343.471,-107.245,173.814,36.270,156.817
C05322=1059.556,343.224,-107.208,173.810,36.265,156.816
C05323=1059.549,342.975,-107.173,173.807,36.260,156.815
C05324=1059.542,342.728,-107.136,173.802,36.255,156.814
C05325=1059.535,342.481,-107.101,173.798,36.251,156.813
C05326=1059.528,342.234,-107.065,173.794,36.246,156.811
C05327=1059.522,341.986,-107.029,173.790,36.241,156.810
C05328=1059.515,341.739,-106.994,173.787,36.236,156.809
C05329=1059.508,341.492,-106.958,173.782,36.231,156.808
C05330=1059.502,341.245,-106.922,173.778,36.226,156.807
C05331=1059.495,340.997,-106.887,173.774,36.222,156.806
C05332=1059.488,340.750,-106.850,173.770,36.217,156.805
C05333=1059.481,340.502,-106.815,173.767,36.212,156.804
C05334=1059.474,340.255,-106.780,173.762,36.207,156.803
C05335=1059.468,340.008,-106.743,173.758,36.203,156.802
C05336=1059.461,339.761,-106.708,173.755,36.197,156.801
C05337=1059.454,339.513,-106.673,173.750,36.193,156.800
C05338=1059.447,339.265,-106.636,173.746,36.188,156.798
C05339=1059.441,339.018,-106.601,173.743,36.183,156.797
C05340=1059.434,338.771,-106.566,173.738,36.179,156.796
C05341=1059.428,338.523,-106.530,173.735,36.174,156.795
C05342=1059.421,338.276,-106.494,173.731,36.169,156.794
C05343=1059.414,338.029,-106.459,173.727,36.164,156.793
C05344=1059.408,337.781,-106.424,173.723,36.159,156.792
C05345=1059.401,337.534,-106.388,173.719,36.155,156.791
C05346=1059.395,337.286,-106.353,173.715,36.150,156.790
C05347=1059.388,337.039,-106.318,173.711,36.145,156.789
C05348=1059.382,336.791,-106.282,173.708,36.141,156.788
C05349=1059.375,336.544,-106.247,173.703,36.136,156.787
C05350=1059.368,336.296,-106.212,173.700,36.131,156.786
C05351=1059.361,336.049,-106.176,173.696,36.126,156.785
C05352=1059.354,335.802,-106.141,173.692,36.122,156.784
C05353=1059.347,335.554,-106.106,173.688,36.117,156.783
C05354=1059.341,335.307,-106.071,173.684,36.113,156.782
C05355=1059.334,335.059,-106.036,173.681,36.108,156.781
C05356=1059.327,334.812,-106.001,173.676,36.104,156.779
C05357=1059.321,334.564,-105.965,173.673,36.099,156.778
C05358=1059.314,334.317,-105.930,173.669,36.094,156.777
C05359=1059.307,334.069,-105.895,173.666,36.090,156.776
C05360=1059.301,333.822,-105.860,173.661,36.085,156.775
C05361=1059.294,333.575,-105.825,173.657,36.080,156.774
C05362=1059.287,333.327,-105.790,173.654,36.076,156.773
C05363=1059.281,333.080,-105.755,173.650,36.071,156.772
C05364=1059.274,332.833,-105.720,173.646,36.066,156.771
C05365=1059.268,332.585,-105.685,173.642,36.062,156.770
C05366=1059.262,332.339,-105.650,173.639,36.057,156.769
C05367=1059.255,332.091,-105.615,173.635,36.053,156.768
C05368=1059.248,331.844,-105.580,173.632,36.048,156.767
C05369=1059.240,331.597,-105.546,173.627,36.044,156.766
C05370=1059.235,331.350,-105.512,173.624,36.039,156.765
C05371=1059.228,331.102,-105.476,173.620,36.034,156.764
C05372=1059.221,330.855,-105.441,173.617,36.030,156.763
C05373=1059.215,330.607,-105.407,173.612,36.025,156.762
C05374=1059.208,330.360,-105.372,173.608,36.021,156.761
C05375=1059.201,330.112,-105.337,173.605,36.017,156.760
C05376=1059.195,329.865,-105.303,173.601,36.012,156.759
C05377=1059.188,329.617,-105.269,173.598,36.007,156.758
C05378=1059.181,329.370,-105.234,173.593,36.003,156.757
C05379=1059.175,329.122,-105.199,173.590,35.999,156.756
C05380=1059.167,328.875,-105.165,173.586,35.994,156.755
C05381=1059.161,328.627,-105.130,173.583,35.990,156.754
C05382=1059.154,328.379,-105.095,173.579,35.986,156.753
C05383=1059.147,328.132,-105.061,173.575,35.981,156.752
C05384=1059.141,327.884,-105.027,173.571,35.977,156.751
C05385=1059.134,327.637,-104.992,173.568,35.972,156.750
C05386=1059.127,327.389,-104.958,173.564,35.968,156.749
C05387=1059.121,327.141,-104.924,173.561,35.963,156.748
C05388=1059.114,326.894,-104.889,173.557,35.959,156.747
C05389=1059.107,326.646,-104.855,173.553,35.955,156.746
C05390=1059.101,326.399,-104.821,173.549,35.951,156.746
C05391=1059.094,326.151,-104.786,173.546,35.946,156.745
C05392=1059.087,325.904,-104.752,173.542,35.941,156.744
C05393=1059.080,325.656,-104.717,173.539,35.937,156.743
C05394=1059.074,325.409,-104.684,173.535,35.933,156.742
C05395=1059.067,325.161,-104.650,173.532,35.929,156.741
C05396=1059.061,324.913,-104.615,173.527,35.924,156.740
C05397=1059.054,324.665,-104.581,173.524,35.920,156.739
C05398=1059.047,324.419,-104.547,173.521,35.916,156.738
C05399=1059.040,324.171,-104.513,173.517,35.911,156.737
C05400=1059.034,323.923,-104.478,173.514,35.907,156.736
C05401=1059.028,323.676,-104.444,173.510,35.902,156.735
C05402=1059.021,323.428,-104.410,173.507,35.898,156.734
C05403=1059.014,323.180,-104.376,173.503,35.894,156.733
C05404=1059.008,322.933,-104.343,173.500,35.890,156.732
C05405=1059.001,322.685,-104.308,173.495,35.885,156.731
C05406=1058.995,322.437,-104.274,173.492,35.881,156.730
C05407=1058.988,322.190,-104.240,173.488,35.876,156.729
C05408=1058.982,321.942,-104.206,173.485,35.872,156.728
C05409=1058.975,321.695,-104.172,173.481,35.868,156.727
C05410=1058.969,321.447,-104.138,173.478,35.864,156.726
C05411=1058.961,321.200,-104.104,173.474,35.859,156.725
C05412=1058.956,320.952,-104.070,173.471,35.855,156.725
C05413=1058.948,320.705,-104.036,173.467,35.851,156.724
C05414=1058.943,320.457,-104.003,173.464,35.846,156.723
C05415=1058.936,320.209,-103.968,173.460,35.842,156.722
C05416=1058.930,319.962,-103.935,173.457,35.838,156.721
C05417=1058.923,319.714,-103.901,173.454,35.833,156.720
C05418=1058.917,319.467,-103.867,173.450,35.829,156.719
C05419=1058.910,319.219,-103.833,173.447,35.825,156.718
C05420=1058.904,318.971,-103.800,173.443,35.821,156.717
C05421=1058.897,318.723,-103.766,173.440,35.816,156.716
